              sync()
            end
            $ 440 "MoveJ"
            $ 441 "Zona_izq1" "breakAfter"
            movej(get_inverse_kin(Zona_izq1_p, qnear=Zona_izq1_q), a=1.3962634015954636, v=1.0471975511965976)
            $ 442 "Posicion_Cero" "breakAfter"
            movej(get_inverse_kin(Posicion_Cero_p, qnear=Posicion_Cero_q), a=1.3962634015954636, v=1.0471975511965976)
            $ 443 "Call Quitar_Broca_Chida"
            Quitar_Broca_Chida()
            $ 444 "Set carrusel_home=Encender"
            modbus_set_output_signal("carrusel_home", True)
            $ 445 "Wait: 1.0"
            sleep(1.0)
            $ 446 "Set carrusel_home=Apagar"
            modbus_set_output_signal("carrusel_home", False)
            $ 447 "Set mensaje_mw10=70"
            modbus_set_output_register("mensaje_mw10", 70)
            $ 448 "Wait Continuar_M30=HI"
            while (modbus_get_signal_status("Continuar_M30") == False):
              sync()
            end
            $ 449 "Wait: 1.0"
            sleep(1.0)
            $ 450 "Set mensaje_mw10=120"
            modbus_set_output_register("mensaje_mw10", 120)
            $ 451 "Wait Continuar_M30=HI"
            while (modbus_get_signal_status("Continuar_M30") == False):
              sync()
            end
            $ 452 "Wait: 1.0"
            sleep(1.0)
            $ 453 "Set carrusel_home=Encender"
            modbus_set_output_signal("carrusel_home", True)
            $ 454 "Wait: 1.0"
            sleep(1.0)
            $ 455 "Set carrusel_home=Apagar"
            modbus_set_output_signal("carrusel_home", False)
            $ 456 "Set mensaje_mw10=75"
            modbus_set_output_register("mensaje_mw10", 75)
            $ 457 "Wait Continuar_M30=HI"
            while (modbus_get_signal_status("Continuar_M30") == False):
              sync()
            end
            $ 458 "Wait: 1.0"
            sleep(1.0)
            $ 459 "Call Poner_Broca"
            Poner_Broca()
            $ 460 "broca≔1935"
            global broca=1935
            $ 461 "MoveJ"
            $ 462 "Posicion_Cero" "breakAfter"
            movej(get_inverse_kin(Posicion_Cero_p, qnear=Posicion_Cero_q), a=1.3962634015954636, v=1.0471975511965976)
            $ 463 "Zona_izq1" "breakAfter"
            movej(get_inverse_kin(Zona_izq1_p, qnear=Zona_izq1_q), a=1.3962634015954636, v=1.0471975511965976)
            $ 464 "Set mensaje_mw10=80"
            modbus_set_output_register("mensaje_mw10", 80)
            $ 465 "Wait Continuar_M30=HI"
            while (modbus_get_signal_status("Continuar_M30") == False):
              sync()
            end
            $ 466 "Wait: 1.0"
            sleep(1.0)
            $ 467 "Set mensaje_mw10=150"
            modbus_set_output_register("mensaje_mw10", 150)
            $ 468 "Wait Continuar_M30=HI"
            while (modbus_get_signal_status("Continuar_M30") == False):
              sync()
            end
            $ 469 "Wait: 1.0"
            sleep(1.0)
          end
        end
        $ 470 "barrenoActual≔barrenoActual+1"
        global barrenoActual=barrenoActual+1
      end
      $ 471 "Linea 1 a 1935"
      $ 472 "broca≔1935"
      global broca=1935
      $ 473 "Buje_inicial"
      $ 474 "Buje_Inicial≔L1B2"
      global Buje_Inicial=L1B2
      $ 475 "Buje_final"
      $ 476 "Buje_Final≔L1B1"
      global Buje_Final=L1B1
      $ 477 "barrenosTotales≔27"
      global barrenosTotales=27
      $ 478 "barrenoActual≔1"
      global barrenoActual=1
      $ 479 "Loop barrenoActual≤barrenosTotales"
      while (barrenoActual <= barrenosTotales):
        $ 480 "MoveL"
        $ 481 "bajada_broca≔p[0,0,0.009,0,0,0]"
        global bajada_broca=p[0,0,0.009,0,0,0]
        $ 482 "internos≔interpolate_pose(Buje_Inicial, Buje_Final, ((barrenoActual)-1)/((barrenosTotales)-1))"
        global internos= interpolate_pose (Buje_Inicial, Buje_Final, ((barrenoActual)-1)/((barrenosTotales)-1))
        $ 483 "Alturas"
        $ 484 "If barrenoActual≟3 or barrenoActual≟5 or barrenoActual≟7 or barrenoActual≟9 or barrenoActual≟11 or barrenoActual≟13 or barrenoActual≟15 or barrenoActual≟17 or barrenoActual≟19 or barrenoActual≟21 or barrenoActual≟23 or barrenoActual≟25 or barrenoActual≟27 or barrenoActual≟1"
        if (barrenoActual == 3  or  barrenoActual == 5  or  barrenoActual == 7  or  barrenoActual == 9  or  barrenoActual == 11  or  barrenoActual == 13  or  barrenoActual == 15  or  barrenoActual == 17  or  barrenoActual == 19  or  barrenoActual == 21  or  barrenoActual == 23  or  barrenoActual == 25  or  barrenoActual == 27  or  barrenoActual == 1):
          $ 485 "Set mensaje_mw10=200"
          modbus_set_output_register("mensaje_mw10", 200)
          $ 486 "Wait Continuar_M30=HI"
          while (modbus_get_signal_status("Continuar_M30") == False):
            sync()
          end
          $ 487 "Wait: 1.0"
          sleep(1.0)
          $ 488 "Set mensaje_mw10=150"
          modbus_set_output_register("mensaje_mw10", 150)
          $ 489 "Wait: 1.0"
          sleep(1.0)
        end
        $ 490 "MoveJ"
        $ 491 "internos" "breakAfter"
        movej(internos, a=1.3962634015954636, v=1.0471975511965976)
        $ 492 "Wait: 2.0"
        sleep(2.0)
        $ 493 "If P1h[2]<P2h[2]"
        if (P1h[2]<P2h[2]):
          $ 494 "acomodin≔(altura/(barrenosTotales-1))*(barrenoActual-1)"
          global acomodin=(altura/(barrenosTotales-1))*(barrenoActual-1)
          $ 495 "tcp_chido≔get_actual_tcp_pose()"
          global tcp_chido= get_actual_tcp_pose ()
          $ 496 "offset_bajada≔p[tcp_chido[0],tcp_chido[1],((alta-0.0095)-(acomodin/1000)),tcp_chido[3],tcp_chido[4],tcp_chido[5]]"
          global offset_bajada=p[tcp_chido[0],tcp_chido[1],((alta-0.0095)-(acomodin/1000)),tcp_chido[3],tcp_chido[4],tcp_chido[5]]
          $ 497 "MoveL"
          $ 498 "offset_bajada" "breakAfter"
          movel(offset_bajada, a=0.03, v=0.015)
        else:
          $ 499 "Else" "noBreak"
          $ 500 "acomodin≔(altura/(barrenosTotales-1))*(26-(barrenoActual-1))"
          global acomodin=(altura/(barrenosTotales-1))*(26-(barrenoActual-1))
          $ 501 "tcp_chido≔get_actual_tcp_pose()"
          global tcp_chido= get_actual_tcp_pose ()
          $ 502 "offset_bajada≔p[tcp_chido[0],tcp_chido[1],((alta-0.0095)-(acomodin/1000)),tcp_chido[3],tcp_chido[4],tcp_chido[5]]"
          global offset_bajada=p[tcp_chido[0],tcp_chido[1],((alta-0.0095)-(acomodin/1000)),tcp_chido[3],tcp_chido[4],tcp_chido[5]]
          $ 503 "MoveL"
          $ 504 "offset_bajada" "breakAfter"
          movel(offset_bajada, a=0.03, v=0.015)
        end
        $ 505 "Freemove"
        $ 506 "Wait: 2.0"
        sleep(2.0)
        $ 507 "freedrive_mode()"
        freedrive_mode()
        $ 508 "Wait: 2.5"
        sleep(2.5)
        $ 509 "end_freedrive_mode()"
        end_freedrive_mode()
        $ 510 "Wait: 0.3"
        sleep(0.3)
        $ 511 "Set CO[1]=Encender"
        set_configurable_digital_out(1, True)
        $ 512 "Wait: 1.0"
        sleep(1.0)
        $ 513 "Wait: 0.3"
        sleep(0.3)
        $ 514 "Wait: 0.3"
        sleep(0.3)
        $ 515 "Wait: 0.3"
        sleep(0.3)
        $ 516 "Loop 2 times"
        Loop_15 = 0
        while (Loop_15 < 2):
          $ 517 "Poses_taladrado≔pose_sub(get_actual_tcp_pose(), bajada_broca)"
          global Poses_taladrado= pose_sub ( get_actual_tcp_pose (), bajada_broca)
          $ 518 "Poses_taladrado" "breakAfter"
          movel(Poses_taladrado, a=0.005, v=0.001)
          $ 519 "If bajada_broca≟p[0,0,0.018,0,0,0]"
          if (bajada_broca == p[0,0,0.018,0,0,0]):
            $ 520 "num_barreno≔str_cat('Barreno: ',barrenoActual)"
            global num_barreno=str_cat("Barreno: ",barrenoActual)
            $ 521 "tcp_actual≔get_actual_tcp_pose()"
            global tcp_actual= get_actual_tcp_pose ()
            $ 522 "X_actual≔str_cat('     X: ',tcp_actual[0])"
            global X_actual=str_cat("     X: ",tcp_actual[0])
            $ 523 "Y_actual≔str_cat('     Y: ',tcp_actual[1])"
            global Y_actual=str_cat("     Y: ",tcp_actual[1])
            $ 524 "pos_barreno≔str_cat(X_actual,Y_actual)"
            global pos_barreno=str_cat(X_actual,Y_actual)
            $ 525 "textmsg(num_barreno,pos_barreno)"
            textmsg(num_barreno,pos_barreno)
          end
          $ 526 "Poses_taladrado≔pose_add(get_actual_tcp_pose(), bajada_broca)"
          global Poses_taladrado= pose_add ( get_actual_tcp_pose (), bajada_broca)
          $ 527 "Poses_taladrado" "breakAfter"
          movel(Poses_taladrado, a=0.01, v=0.01)
          $ 528 "bajada_broca≔pose_add(bajada_broca, p[0,0,0.009,0,0,0])"
          global bajada_broca= pose_add (bajada_broca, p[0,0,0.009,0,0,0])
          Loop_15 = Loop_15 + 1
        end
        $ 529 "Direction: Base Z+"
        global move_thread_flag_529=0
        thread move_thread_529():
          enter_critical
          move_thread_flag_529 = 1
          local towardsPos=calculate_point_to_move_towards(p[0.0,0.0,0.0,0.0,0.0,0.0], [0.0,0.0,1.0], 0.05)
          movel(towardsPos, a=0.04, v=0.03)
          move_thread_flag_529 = 2
          exit_critical
        end
        move_thread_flag_529 = 0
        move_thread_han_529 = run move_thread_529()
        while (True):
          sleep(1.0E-10)
          if (move_thread_flag_529 > 1):
            join move_thread_han_529
            $ 530 "Until (distance)"
            break
          end
          sync()
        end
        $ 531 "MoveJ"
        $ 532 "internos" "breakAfter"
        movej(internos, a=1.3962634015954636, v=1.0471975511965976)
        $ 533 "Wait: 0.3"
        sleep(0.3)
        $ 534 "Set CO[1]=Apagar"
        set_configurable_digital_out(1, False)
        $ 535 "Wait: 0.3"
        sleep(0.3)
        $ 536 "If barrenoActual≟13 or barrenoActual≟27"
        if (barrenoActual == 13  or  barrenoActual == 27):
          $ 537 "Direction: Base Z+"
          global move_thread_flag_537=0
          thread move_thread_537():
            enter_critical
            move_thread_flag_537 = 1
            local towardsPos=calculate_point_to_move_towards(p[0.0,0.0,0.0,0.0,0.0,0.0], [0.0,0.0,1.0], 0.03)
            movel(towardsPos, a=1.2, v=0.25)
            move_thread_flag_537 = 2
            exit_critical
          end
          move_thread_flag_537 = 0
          move_thread_han_537 = run move_thread_537()
          while (True):
            sleep(1.0E-10)
            if (move_thread_flag_537 > 1):
              join move_thread_han_537
              $ 538 "Until (distance)"
              break
            end
            sync()
          end
          $ 539 "MoveJ"
          $ 540 "Zona_izq1" "breakAfter"
          movej(get_inverse_kin(Zona_izq1_p, qnear=Zona_izq1_q), a=1.3962634015954636, v=1.0471975511965976)
          $ 541 "Posicion_Cero" "breakAfter"
          movej(get_inverse_kin(Posicion_Cero_p, qnear=Posicion_Cero_q), a=1.3962634015954636, v=1.0471975511965976)
          $ 542 "Call Quitar_Broca_Chida"
          Quitar_Broca_Chida()
          $ 543 "Call Poner_Broca"
          Poner_Broca()
          $ 544 "MoveJ"
          $ 545 "Posicion_Cero" "breakAfter"
          movej(get_inverse_kin(Posicion_Cero_p, qnear=Posicion_Cero_q), a=1.3962634015954636, v=1.0471975511965976)
          $ 546 "Zona_izq1" "breakAfter"
          movej(get_inverse_kin(Zona_izq1_p, qnear=Zona_izq1_q), a=1.3962634015954636, v=1.0471975511965976)
        end
        $ 547 "barrenoActual≔barrenoActual+1"
        global barrenoActual=barrenoActual+1
      end
      $ 548 "Linea 2 a 1935"
      $ 549 "broca≔1935"
      global broca=1935
      $ 550 "Buje_inicial"
      $ 551 "Buje_Inicial≔L2B2"
      global Buje_Inicial=L2B2
      $ 552 "Buje_final"
      $ 553 "Buje_Final≔L2B1"
      global Buje_Final=L2B1
      $ 554 "barrenosTotales≔27"
      global barrenosTotales=27
      $ 555 "barrenoActual≔1"
      global barrenoActual=1
      $ 556 "Loop barrenoActual≤barrenosTotales"
      while (barrenoActual <= barrenosTotales):
        $ 557 "MoveL"
        $ 558 "bajada_broca≔p[0,0,0.009,0,0,0]"
        global bajada_broca=p[0,0,0.009,0,0,0]
        $ 559 "internos≔interpolate_pose(Buje_Inicial, Buje_Final, ((barrenoActual)-1)/((barrenosTotales)-1))"
        global internos= interpolate_pose (Buje_Inicial, Buje_Final, ((barrenoActual)-1)/((barrenosTotales)-1))
        $ 560 "Alturas"
        $ 561 "If barrenoActual≟3 or barrenoActual≟5 or barrenoActual≟7 or barrenoActual≟9 or barrenoActual≟11 or barrenoActual≟13 or barrenoActual≟15 or barrenoActual≟17 or barrenoActual≟19 or barrenoActual≟21 or barrenoActual≟23 or barrenoActual≟25 or barrenoActual≟27 or barrenoActual≟1"
        if (barrenoActual == 3  or  barrenoActual == 5  or  barrenoActual == 7  or  barrenoActual == 9  or  barrenoActual == 11  or  barrenoActual == 13  or  barrenoActual == 15  or  barrenoActual == 17  or  barrenoActual == 19  or  barrenoActual == 21  or  barrenoActual == 23  or  barrenoActual == 25  or  barrenoActual == 27  or  barrenoActual == 1):
          $ 562 "Set mensaje_mw10=200"
          modbus_set_output_register("mensaje_mw10", 200)
          $ 563 "Wait Continuar_M30=HI"
          while (modbus_get_signal_status("Continuar_M30") == False):
            sync()
          end
          $ 564 "Wait: 1.0"
          sleep(1.0)
          $ 565 "Set mensaje_mw10=150"
          modbus_set_output_register("mensaje_mw10", 150)
          $ 566 "Wait: 1.0"
          sleep(1.0)
        end
        $ 567 "MoveJ"
        $ 568 "internos" "breakAfter"
        movej(internos, a=1.3962634015954636, v=1.0471975511965976)
        $ 569 "Wait: 2.0"
        sleep(2.0)
        $ 570 "If P1h[2]<P2h[2]"
        if (P1h[2]<P2h[2]):
          $ 571 "acomodin≔(altura/(barrenosTotales-1))*(barrenoActual-1)"
          global acomodin=(altura/(barrenosTotales-1))*(barrenoActual-1)
          $ 572 "tcp_chido≔get_actual_tcp_pose()"
          global tcp_chido= get_actual_tcp_pose ()
          $ 573 "offset_bajada≔p[tcp_chido[0],tcp_chido[1],((alta-0.0095)-(acomodin/1000)),tcp_chido[3],tcp_chido[4],tcp_chido[5]]"
          global offset_bajada=p[tcp_chido[0],tcp_chido[1],((alta-0.0095)-(acomodin/1000)),tcp_chido[3],tcp_chido[4],tcp_chido[5]]
          $ 574 "MoveL"
          $ 575 "offset_bajada" "breakAfter"
          movel(offset_bajada, a=0.03, v=0.015)
        else:
          $ 576 "Else" "noBreak"
          $ 577 "acomodin≔(altura/(barrenosTotales-1))*(26-(barrenoActual-1))"
          global acomodin=(altura/(barrenosTotales-1))*(26-(barrenoActual-1))
          $ 578 "tcp_chido≔get_actual_tcp_pose()"
          global tcp_chido= get_actual_tcp_pose ()
          $ 579 "offset_bajada≔p[tcp_chido[0],tcp_chido[1],((alta-0.0095)-(acomodin/1000)),tcp_chido[3],tcp_chido[4],tcp_chido[5]]"
          global offset_bajada=p[tcp_chido[0],tcp_chido[1],((alta-0.0095)-(acomodin/1000)),tcp_chido[3],tcp_chido[4],tcp_chido[5]]
          $ 580 "MoveL"
          $ 581 "offset_bajada" "breakAfter"
          movel(offset_bajada, a=0.03, v=0.015)
        end
        $ 582 "Freemove"
        $ 583 "Wait: 2.0"
        sleep(2.0)
        $ 584 "freedrive_mode()"
        freedrive_mode()
        $ 585 "Wait: 2.5"
        sleep(2.5)
        $ 586 "end_freedrive_mode()"
        end_freedrive_mode()
        $ 587 "Wait: 0.3"
        sleep(0.3)
        $ 588 "Set CO[1]=Encender"
        set_configurable_digital_out(1, True)
        $ 589 "Wait: 1.0"
        sleep(1.0)
        $ 590 "Wait: 0.3"
        sleep(0.3)
        $ 591 "Wait: 0.3"
        sleep(0.3)
        $ 592 "Wait: 0.3"
        sleep(0.3)
        $ 593 "Loop 2 times"
        Loop_17 = 0
        while (Loop_17 < 2):
          $ 594 "Poses_taladrado≔pose_sub(get_actual_tcp_pose(), bajada_broca)"
          global Poses_taladrado= pose_sub ( get_actual_tcp_pose (), bajada_broca)
          $ 595 "Poses_taladrado" "breakAfter"
          movel(Poses_taladrado, a=0.005, v=0.001)
          $ 596 "If bajada_broca≟p[0,0,0.018,0,0,0]"
          if (bajada_broca == p[0,0,0.018,0,0,0]):
            $ 597 "num_barreno≔str_cat('Barreno: ',barrenoActual)"
            global num_barreno=str_cat("Barreno: ",barrenoActual)
            $ 598 "tcp_actual≔get_actual_tcp_pose()"
            global tcp_actual= get_actual_tcp_pose ()
            $ 599 "X_actual≔str_cat('     X: ',tcp_actual[0])"
            global X_actual=str_cat("     X: ",tcp_actual[0])
            $ 600 "Y_actual≔str_cat('     Y: ',tcp_actual[1])"
            global Y_actual=str_cat("     Y: ",tcp_actual[1])
            $ 601 "pos_barreno≔str_cat(X_actual,Y_actual)"
            global pos_barreno=str_cat(X_actual,Y_actual)
            $ 602 "textmsg(num_barreno,pos_barreno)"
            textmsg(num_barreno,pos_barreno)
          end
          $ 603 "Poses_taladrado≔pose_add(get_actual_tcp_pose(), bajada_broca)"
          global Poses_taladrado= pose_add ( get_actual_tcp_pose (), bajada_broca)
          $ 604 "Poses_taladrado" "breakAfter"
          movel(Poses_taladrado, a=0.01, v=0.01)
          $ 605 "bajada_broca≔pose_add(bajada_broca, p[0,0,0.009,0,0,0])"
          global bajada_broca= pose_add (bajada_broca, p[0,0,0.009,0,0,0])
          Loop_17 = Loop_17 + 1
        end
        $ 606 "Direction: Base Z+"
        global move_thread_flag_606=0
        thread move_thread_606():
          enter_critical
          move_thread_flag_606 = 1
          local towardsPos=calculate_point_to_move_towards(p[0.0,0.0,0.0,0.0,0.0,0.0], [0.0,0.0,1.0], 0.05)
          movel(towardsPos, a=0.04, v=0.03)
          move_thread_flag_606 = 2
          exit_critical
        end
        move_thread_flag_606 = 0
        move_thread_han_606 = run move_thread_606()
        while (True):
          sleep(1.0E-10)
          if (move_thread_flag_606 > 1):
            join move_thread_han_606
            $ 607 "Until (distance)"
            break
          end
          sync()
        end
        $ 608 "MoveJ"
        $ 609 "internos" "breakAfter"
        movej(internos, a=1.3962634015954636, v=1.0471975511965976)
        $ 610 "Wait: 0.3"
        sleep(0.3)
        $ 611 "Set CO[1]=Apagar"
        set_configurable_digital_out(1, False)
        $ 612 "Wait: 0.3"
        sleep(0.3)
        $ 613 "If barrenoActual≟13"
        if (barrenoActual == 13):
          $ 614 "Direction: Base Z+"
          global move_thread_flag_614=0
          thread move_thread_614():
            enter_critical
            move_thread_flag_614 = 1
            local towardsPos=calculate_point_to_move_towards(p[0.0,0.0,0.0,0.0,0.0,0.0], [0.0,0.0,1.0], 0.03)
            movel(towardsPos, a=1.2, v=0.25)
            move_thread_flag_614 = 2
            exit_critical
          end
          move_thread_flag_614 = 0
          move_thread_han_614 = run move_thread_614()
          while (True):
            sleep(1.0E-10)
            if (move_thread_flag_614 > 1):
              join move_thread_han_614
              $ 615 "Until (distance)"
              break
            end
            sync()
          end
          $ 616 "MoveJ"
          $ 617 "Zona_izq1" "breakAfter"
          movej(get_inverse_kin(Zona_izq1_p, qnear=Zona_izq1_q), a=1.3962634015954636, v=1.0471975511965976)
          $ 618 "Posicion_Cero" "breakAfter"
          movej(get_inverse_kin(Posicion_Cero_p, qnear=Posicion_Cero_q), a=1.3962634015954636, v=1.0471975511965976)
          $ 619 "Call Quitar_Broca_Chida"
          Quitar_Broca_Chida()
          $ 620 "Call Poner_Broca"
          Poner_Broca()
          $ 621 "MoveJ"
          $ 622 "Posicion_Cero" "breakAfter"
          movej(get_inverse_kin(Posicion_Cero_p, qnear=Posicion_Cero_q), a=1.3962634015954636, v=1.0471975511965976)
          $ 623 "Zona_izq1" "breakAfter"
          movej(get_inverse_kin(Zona_izq1_p, qnear=Zona_izq1_q), a=1.3962634015954636, v=1.0471975511965976)
        else:
          $ 624 "ElseIf barrenoActual≟27"
          if (barrenoActual == 27):
            $ 625 "Direction: Base Z+"
            global move_thread_flag_625=0
            thread move_thread_625():
              enter_critical
              move_thread_flag_625 = 1
              local towardsPos=calculate_point_to_move_towards(p[0.0,0.0,0.0,0.0,0.0,0.0], [0.0,0.0,1.0], 0.03)
              movel(towardsPos, a=1.2, v=0.25)
              move_thread_flag_625 = 2
              exit_critical
            end
            move_thread_flag_625 = 0
            move_thread_han_625 = run move_thread_625()
            while (True):
              sleep(1.0E-10)
              if (move_thread_flag_625 > 1):
                join move_thread_han_625
                $ 626 "Until (distance)"
                break
              end
              sync()
            end
            $ 627 "MoveJ"
            $ 628 "Zona_izq1" "breakAfter"
            movej(get_inverse_kin(Zona_izq1_p, qnear=Zona_izq1_q), a=1.3962634015954636, v=1.0471975511965976)
            $ 629 "Posicion_Cero" "breakAfter"
            movej(get_inverse_kin(Posicion_Cero_p, qnear=Posicion_Cero_q), a=1.3962634015954636, v=1.0471975511965976)
            $ 630 "Call Quitar_Broca_Chida"
            Quitar_Broca_Chida()
            $ 631 "Set carrusel_home=Encender"
            modbus_set_output_signal("carrusel_home", True)
            $ 632 "Wait: 1.0"
            sleep(1.0)
            $ 633 "Set carrusel_home=Apagar"
            modbus_set_output_signal("carrusel_home", False)
            $ 634 "Set mensaje_mw10=85"
            modbus_set_output_register("mensaje_mw10", 85)
            $ 635 "Wait Continuar_M30=HI"
            while (modbus_get_signal_status("Continuar_M30") == False):
              sync()
            end
            $ 636 "Wait: 1.0"
            sleep(1.0)
            $ 637 "Set mensaje_mw10=120"
            modbus_set_output_register("mensaje_mw10", 120)
            $ 638 "Wait Continuar_M30=HI"
            while (modbus_get_signal_status("Continuar_M30") == False):
              sync()
            end
            $ 639 "Wait: 1.0"
            sleep(1.0)
            $ 640 "Set carrusel_home=Encender"
            modbus_set_output_signal("carrusel_home", True)
            $ 641 "Wait: 1.0"
            sleep(1.0)
            $ 642 "Set carrusel_home=Apagar"
            modbus_set_output_signal("carrusel_home", False)
            $ 643 "Set mensaje_mw10=90"
            modbus_set_output_register("mensaje_mw10", 90)
            $ 644 "Wait Continuar_M30=HI"
            while (modbus_get_signal_status("Continuar_M30") == False):
              sync()
            end
            $ 645 "Wait: 1.0"
            sleep(1.0)
            $ 646 "Call Poner_Broca"
            Poner_Broca()
            $ 647 "broca≔217"
            global broca=217
            $ 648 "MoveJ"
            $ 649 "Posicion_Cero" "breakAfter"
            movej(get_inverse_kin(Posicion_Cero_p, qnear=Posicion_Cero_q), a=1.3962634015954636, v=1.0471975511965976)
            $ 650 "Zona_izq1" "breakAfter"
            movej(get_inverse_kin(Zona_izq1_p, qnear=Zona_izq1_q), a=1.3962634015954636, v=1.0471975511965976)
            $ 651 "Set mensaje_mw10=95"
            modbus_set_output_register("mensaje_mw10", 95)
            $ 652 "Wait Continuar_M30=HI"
            while (modbus_get_signal_status("Continuar_M30") == False):
              sync()
            end
            $ 653 "Wait: 1.0"
            sleep(1.0)
            $ 654 "Set mensaje_mw10=150"
            modbus_set_output_register("mensaje_mw10", 150)
            $ 655 "Wait Continuar_M30=HI"
            while (modbus_get_signal_status("Continuar_M30") == False):
              sync()
            end
            $ 656 "Wait: 1.0"
            sleep(1.0)
          end
        end
        $ 657 "barrenoActual≔barrenoActual+1"
        global barrenoActual=barrenoActual+1
      end
      $ 658 "Linea 1 a 217"
      $ 659 "broca≔217"
      global broca=217
      $ 660 "Buje_inicial"
      $ 661 "Buje_Inicial≔L1B2"
      global Buje_Inicial=L1B2
      $ 662 "Buje_final"
      $ 663 "Buje_Final≔L1B1"
      global Buje_Final=L1B1
      $ 664 "barrenosTotales≔27"
      global barrenosTotales=27
      $ 665 "barrenoActual≔1"
      global barrenoActual=1
      $ 666 "Loop barrenoActual≤barrenosTotales"
      while (barrenoActual <= barrenosTotales):
        $ 667 "MoveL"
        $ 668 "bajada_broca≔p[0,0,0.018,0,0,0]"
        global bajada_broca=p[0,0,0.018,0,0,0]
        $ 669 "internos≔interpolate_pose(Buje_Inicial, Buje_Final, ((barrenoActual)-1)/((barrenosTotales)-1))"
        global internos= interpolate_pose (Buje_Inicial, Buje_Final, ((barrenoActual)-1)/((barrenosTotales)-1))
        $ 670 "Alturas"
        $ 671 "If barrenoActual≟3 or barrenoActual≟5 or barrenoActual≟7 or barrenoActual≟9 or barrenoActual≟11 or barrenoActual≟13 or barrenoActual≟15 or barrenoActual≟17 or barrenoActual≟19 or barrenoActual≟21 or barrenoActual≟23 or barrenoActual≟25 or barrenoActual≟27 or barrenoActual≟1"
        if (barrenoActual == 3  or  barrenoActual == 5  or  barrenoActual == 7  or  barrenoActual == 9  or  barrenoActual == 11  or  barrenoActual == 13  or  barrenoActual == 15  or  barrenoActual == 17  or  barrenoActual == 19  or  barrenoActual == 21  or  barrenoActual == 23  or  barrenoActual == 25  or  barrenoActual == 27  or  barrenoActual == 1):
          $ 672 "Set mensaje_mw10=200"
          modbus_set_output_register("mensaje_mw10", 200)
          $ 673 "Wait Continuar_M30=HI"
          while (modbus_get_signal_status("Continuar_M30") == False):
            sync()
          end
          $ 674 "Wait: 1.0"
          sleep(1.0)
          $ 675 "Set mensaje_mw10=150"
          modbus_set_output_register("mensaje_mw10", 150)
          $ 676 "Wait: 1.0"
          sleep(1.0)
        end
        $ 677 "MoveJ"
        $ 678 "internos" "breakAfter"
        movej(internos, a=1.3962634015954636, v=1.0471975511965976)
        $ 679 "Wait: 2.0"
        sleep(2.0)
        $ 680 "If P1h[2]<P2h[2]"
        if (P1h[2]<P2h[2]):
          $ 681 "acomodin≔(altura/(barrenosTotales-1))*(barrenoActual-1)"
          global acomodin=(altura/(barrenosTotales-1))*(barrenoActual-1)
          $ 682 "tcp_chido≔get_actual_tcp_pose()"
          global tcp_chido= get_actual_tcp_pose ()
          $ 683 "offset_bajada≔p[tcp_chido[0],tcp_chido[1],((alta-0.0095)-(acomodin/1000)),tcp_chido[3],tcp_chido[4],tcp_chido[5]]"
          global offset_bajada=p[tcp_chido[0],tcp_chido[1],((alta-0.0095)-(acomodin/1000)),tcp_chido[3],tcp_chido[4],tcp_chido[5]]
          $ 684 "MoveL"
          $ 685 "offset_bajada" "breakAfter"
          movel(offset_bajada, a=0.03, v=0.015)
        else:
          $ 686 "Else" "noBreak"
          $ 687 "acomodin≔(altura/(barrenosTotales-1))*(26-(barrenoActual-1))"
          global acomodin=(altura/(barrenosTotales-1))*(26-(barrenoActual-1))
          $ 688 "tcp_chido≔get_actual_tcp_pose()"
          global tcp_chido= get_actual_tcp_pose ()
          $ 689 "offset_bajada≔p[tcp_chido[0],tcp_chido[1],((alta-0.0095)-(acomodin/1000)),tcp_chido[3],tcp_chido[4],tcp_chido[5]]"
          global offset_bajada=p[tcp_chido[0],tcp_chido[1],((alta-0.0095)-(acomodin/1000)),tcp_chido[3],tcp_chido[4],tcp_chido[5]]
          $ 690 "MoveL"
          $ 691 "offset_bajada" "breakAfter"
          movel(offset_bajada, a=0.03, v=0.015)
        end
        $ 692 "Freemove"
        $ 693 "Wait: 2.0"
        sleep(2.0)
        $ 694 "freedrive_mode()"
        freedrive_mode()
        $ 695 "Wait: 2.5"
        sleep(2.5)
        $ 696 "end_freedrive_mode()"
        end_freedrive_mode()
        $ 697 "Wait: 0.3"
        sleep(0.3)
        $ 698 "Set CO[1]=Encender"
        set_configurable_digital_out(1, True)
        $ 699 "Wait: 1.0"
        sleep(1.0)
        $ 700 "Wait: 0.3"
        sleep(0.3)
        $ 701 "Wait: 0.3"
        sleep(0.3)
        $ 702 "Wait: 0.3"
        sleep(0.3)
        $ 703 "Loop 1 times"
        Loop_19 = 0
        while (Loop_19 < 1):
          $ 704 "Poses_taladrado≔pose_sub(get_actual_tcp_pose(), bajada_broca)"
          global Poses_taladrado= pose_sub ( get_actual_tcp_pose (), bajada_broca)
          $ 705 "Poses_taladrado" "breakAfter"
          movel(Poses_taladrado, a=0.005, v=0.001)
          $ 706 "If bajada_broca≟p[0,0,0.018,0,0,0]"
          if (bajada_broca == p[0,0,0.018,0,0,0]):
            $ 707 "num_barreno≔str_cat('Barreno: ',barrenoActual)"
            global num_barreno=str_cat("Barreno: ",barrenoActual)
            $ 708 "tcp_actual≔get_actual_tcp_pose()"
            global tcp_actual= get_actual_tcp_pose ()
            $ 709 "X_actual≔str_cat('     X: ',tcp_actual[0])"
            global X_actual=str_cat("     X: ",tcp_actual[0])
            $ 710 "Y_actual≔str_cat('     Y: ',tcp_actual[1])"
            global Y_actual=str_cat("     Y: ",tcp_actual[1])
            $ 711 "pos_barreno≔str_cat(X_actual,Y_actual)"
            global pos_barreno=str_cat(X_actual,Y_actual)
            $ 712 "textmsg(num_barreno,pos_barreno)"
            textmsg(num_barreno,pos_barreno)
          end
          $ 713 "Poses_taladrado≔pose_add(get_actual_tcp_pose(), bajada_broca)"
          global Poses_taladrado= pose_add ( get_actual_tcp_pose (), bajada_broca)
          $ 714 "Poses_taladrado" "breakAfter"
          movel(Poses_taladrado, a=0.01, v=0.01)
          $ 715 "bajada_broca≔pose_add(bajada_broca, p[0,0,0.018,0,0,0])"
          global bajada_broca= pose_add (bajada_broca, p[0,0,0.018,0,0,0])
          Loop_19 = Loop_19 + 1
        end
        $ 716 "Direction: Base Z+"
        global move_thread_flag_716=0
        thread move_thread_716():
          enter_critical
          move_thread_flag_716 = 1
          local towardsPos=calculate_point_to_move_towards(p[0.0,0.0,0.0,0.0,0.0,0.0], [0.0,0.0,1.0], 0.05)
          movel(towardsPos, a=0.04, v=0.03)
          move_thread_flag_716 = 2
          exit_critical
        end
        move_thread_flag_716 = 0
        move_thread_han_716 = run move_thread_716()
        while (True):
          sleep(1.0E-10)
          if (move_thread_flag_716 > 1):
            join move_thread_han_716
            $ 717 "Until (distance)"
            break
          end
          sync()
        end
        $ 718 "MoveJ"
        $ 719 "internos" "breakAfter"
        movej(internos, a=1.3962634015954636, v=1.0471975511965976)
        $ 720 "Wait: 0.3"
        sleep(0.3)
        $ 721 "Set CO[1]=Apagar"
        set_configurable_digital_out(1, False)
        $ 722 "Wait: 0.3"
        sleep(0.3)
        $ 723 "If barrenoActual≟13 or barrenoActual≟27"
        if (barrenoActual == 13  or  barrenoActual == 27):
          $ 724 "Direction: Base Z+"
          global move_thread_flag_724=0
          thread move_thread_724():
            enter_critical
            move_thread_flag_724 = 1
            local towardsPos=calculate_point_to_move_towards(p[0.0,0.0,0.0,0.0,0.0,0.0], [0.0,0.0,1.0], 0.03)
            movel(towardsPos, a=1.2, v=0.25)
            move_thread_flag_724 = 2
            exit_critical
          end
          move_thread_flag_724 = 0
          move_thread_han_724 = run move_thread_724()
          while (True):
            sleep(1.0E-10)
            if (move_thread_flag_724 > 1):
              join move_thread_han_724
              $ 725 "Until (distance)"
              break
            end
            sync()
          end
          $ 726 "MoveJ"
          $ 727 "Zona_izq1" "breakAfter"
          movej(get_inverse_kin(Zona_izq1_p, qnear=Zona_izq1_q), a=1.3962634015954636, v=1.0471975511965976)
          $ 728 "Posicion_Cero" "breakAfter"
          movej(get_inverse_kin(Posicion_Cero_p, qnear=Posicion_Cero_q), a=1.3962634015954636, v=1.0471975511965976)
          $ 729 "Call Quitar_Broca_Chida"
          Quitar_Broca_Chida()
          $ 730 "Call Poner_Broca"
          Poner_Broca()
          $ 731 "MoveJ"
          $ 732 "Posicion_Cero" "breakAfter"
          movej(get_inverse_kin(Posicion_Cero_p, qnear=Posicion_Cero_q), a=1.3962634015954636, v=1.0471975511965976)
          $ 733 "Zona_izq1" "breakAfter"
          movej(get_inverse_kin(Zona_izq1_p, qnear=Zona_izq1_q), a=1.3962634015954636, v=1.0471975511965976)
        end
        $ 734 "barrenoActual≔barrenoActual+1"
        global barrenoActual=barrenoActual+1
      end
      $ 735 "Linea 2 a 217"
      $ 736 "broca≔217"
      global broca=217
      $ 737 "Buje_inicial"
      $ 738 "Buje_Inicial≔L2B2"
      global Buje_Inicial=L2B2
      $ 739 "Buje_final"
      $ 740 "Buje_Final≔L2B1"
      global Buje_Final=L2B1
      $ 741 "barrenosTotales≔27"
      global barrenosTotales=27
      $ 742 "barrenoActual≔1"
      global barrenoActual=1
      $ 743 "Loop barrenoActual≤barrenosTotales"
      while (barrenoActual <= barrenosTotales):
        $ 744 "MoveL"
        $ 745 "bajada_broca≔p[0,0,0.018,0,0,0]"
        global bajada_broca=p[0,0,0.018,0,0,0]
        $ 746 "internos≔interpolate_pose(Buje_Inicial, Buje_Final, ((barrenoActual)-1)/((barrenosTotales)-1))"
        global internos= interpolate_pose (Buje_Inicial, Buje_Final, ((barrenoActual)-1)/((barrenosTotales)-1))
        $ 747 "Alturas"
        $ 748 "If barrenoActual≟3 or barrenoActual≟5 or barrenoActual≟7 or barrenoActual≟9 or barrenoActual≟11 or barrenoActual≟13 or barrenoActual≟15 or barrenoActual≟17 or barrenoActual≟19 or barrenoActual≟21 or barrenoActual≟23 or barrenoActual≟25 or barrenoActual≟27 or barrenoActual≟1"
        if (barrenoActual == 3  or  barrenoActual == 5  or  barrenoActual == 7  or  barrenoActual == 9  or  barrenoActual == 11  or  barrenoActual == 13  or  barrenoActual == 15  or  barrenoActual == 17  or  barrenoActual == 19  or  barrenoActual == 21  or  barrenoActual == 23  or  barrenoActual == 25  or  barrenoActual == 27  or  barrenoActual == 1):
          $ 749 "Set mensaje_mw10=200"
          modbus_set_output_register("mensaje_mw10", 200)
          $ 750 "Wait Continuar_M30=HI"
          while (modbus_get_signal_status("Continuar_M30") == False):
            sync()
          end
          $ 751 "Wait: 1.0"
          sleep(1.0)
          $ 752 "Set mensaje_mw10=150"
          modbus_set_output_register("mensaje_mw10", 150)
          $ 753 "Wait: 1.0"
          sleep(1.0)
        end
        $ 754 "MoveJ"
        $ 755 "internos" "breakAfter"
        movej(internos, a=1.3962634015954636, v=1.0471975511965976)
        $ 756 "Wait: 2.0"
        sleep(2.0)
        $ 757 "If P1h[2]<P2h[2]"
        if (P1h[2]<P2h[2]):
          $ 758 "acomodin≔(altura/(barrenosTotales-1))*(barrenoActual-1)"
          global acomodin=(altura/(barrenosTotales-1))*(barrenoActual-1)
          $ 759 "tcp_chido≔get_actual_tcp_pose()"
          global tcp_chido= get_actual_tcp_pose ()
          $ 760 "offset_bajada≔p[tcp_chido[0],tcp_chido[1],((alta-0.0095)-(acomodin/1000)),tcp_chido[3],tcp_chido[4],tcp_chido[5]]"
          global offset_bajada=p[tcp_chido[0],tcp_chido[1],((alta-0.0095)-(acomodin/1000)),tcp_chido[3],tcp_chido[4],tcp_chido[5]]
          $ 761 "MoveL"
          $ 762 "offset_bajada" "breakAfter"
          movel(offset_bajada, a=0.03, v=0.015)
        else:
          $ 763 "Else" "noBreak"
          $ 764 "acomodin≔(altura/(barrenosTotales-1))*(26-(barrenoActual-1))"
          global acomodin=(altura/(barrenosTotales-1))*(26-(barrenoActual-1))
          $ 765 "tcp_chido≔get_actual_tcp_pose()"
          global tcp_chido= get_actual_tcp_pose ()
          $ 766 "offset_bajada≔p[tcp_chido[0],tcp_chido[1],((alta-0.0095)-(acomodin/1000)),tcp_chido[3],tcp_chido[4],tcp_chido[5]]"
          global offset_bajada=p[tcp_chido[0],tcp_chido[1],((alta-0.0095)-(acomodin/1000)),tcp_chido[3],tcp_chido[4],tcp_chido[5]]
          $ 767 "MoveL"
          $ 768 "offset_bajada" "breakAfter"
          movel(offset_bajada, a=0.03, v=0.015)
        end
        $ 769 "Freemove"
        $ 770 "Wait: 2.0"
        sleep(2.0)
        $ 771 "freedrive_mode()"
        freedrive_mode()
        $ 772 "Wait: 2.5"
        sleep(2.5)
        $ 773 "end_freedrive_mode()"
        end_freedrive_mode()
        $ 774 "Wait: 0.3"
        sleep(0.3)
        $ 775 "Set CO[1]=Encender"
        set_configurable_digital_out(1, True)
        $ 776 "Wait: 1.0"
        sleep(1.0)
        $ 777 "Wait: 0.3"
        sleep(0.3)
        $ 778 "Wait: 0.3"
        sleep(0.3)
        $ 779 "Wait: 0.3"
        sleep(0.3)
        $ 780 "Loop 1 times"
        Loop_21 = 0
        while (Loop_21 < 1):
          $ 781 "Poses_taladrado≔pose_sub(get_actual_tcp_pose(), bajada_broca)"
          global Poses_taladrado= pose_sub ( get_actual_tcp_pose (), bajada_broca)
          $ 782 "Poses_taladrado" "breakAfter"
          movel(Poses_taladrado, a=0.005, v=0.001)
          $ 783 "If bajada_broca≟p[0,0,0.018,0,0,0]"
          if (bajada_broca == p[0,0,0.018,0,0,0]):
            $ 784 "num_barreno≔str_cat('Barreno: ',barrenoActual)"
            global num_barreno=str_cat("Barreno: ",barrenoActual)
            $ 785 "tcp_actual≔get_actual_tcp_pose()"
            global tcp_actual= get_actual_tcp_pose ()
            $ 786 "X_actual≔str_cat('     X: ',tcp_actual[0])"
            global X_actual=str_cat("     X: ",tcp_actual[0])
            $ 787 "Y_actual≔str_cat('     Y: ',tcp_actual[1])"
            global Y_actual=str_cat("     Y: ",tcp_actual[1])
            $ 788 "pos_barreno≔str_cat(X_actual,Y_actual)"
            global pos_barreno=str_cat(X_actual,Y_actual)
            $ 789 "textmsg(num_barreno,pos_barreno)"
            textmsg(num_barreno,pos_barreno)
          end
          $ 790 "Poses_taladrado≔pose_add(get_actual_tcp_pose(), bajada_broca)"
          global Poses_taladrado= pose_add ( get_actual_tcp_pose (), bajada_broca)
          $ 791 "Poses_taladrado" "breakAfter"
          movel(Poses_taladrado, a=0.01, v=0.01)
          $ 792 "bajada_broca≔pose_add(bajada_broca, p[0,0,0.018,0,0,0])"
          global bajada_broca= pose_add (bajada_broca, p[0,0,0.018,0,0,0])
          Loop_21 = Loop_21 + 1
        end
        $ 793 "Direction: Base Z+"
        global move_thread_flag_793=0
        thread move_thread_793():
          enter_critical
          move_thread_flag_793 = 1
          local towardsPos=calculate_point_to_move_towards(p[0.0,0.0,0.0,0.0,0.0,0.0], [0.0,0.0,1.0], 0.05)
          movel(towardsPos, a=0.04, v=0.03)
          move_thread_flag_793 = 2
          exit_critical
        end
        move_thread_flag_793 = 0
        move_thread_han_793 = run move_thread_793()
        while (True):
          sleep(1.0E-10)
          if (move_thread_flag_793 > 1):
            join move_thread_han_793
            $ 794 "Until (distance)"
            break
          end
          sync()
        end
        $ 795 "MoveJ"
        $ 796 "internos" "breakAfter"
        movej(internos, a=1.3962634015954636, v=1.0471975511965976)
        $ 797 "Wait: 0.3"
        sleep(0.3)
        $ 798 "Set CO[1]=Apagar"
        set_configurable_digital_out(1, False)
        $ 799 "Wait: 0.3"
        sleep(0.3)
        $ 800 "If barrenoActual≟13"
        if (barrenoActual == 13):
          $ 801 "Direction: Base Z+"
          global move_thread_flag_801=0
          thread move_thread_801():
            enter_critical
            move_thread_flag_801 = 1
            local towardsPos=calculate_point_to_move_towards(p[0.0,0.0,0.0,0.0,0.0,0.0], [0.0,0.0,1.0], 0.03)
            movel(towardsPos, a=1.2, v=0.25)
            move_thread_flag_801 = 2
            exit_critical
          end
          move_thread_flag_801 = 0
          move_thread_han_801 = run move_thread_801()
          while (True):
            sleep(1.0E-10)
            if (move_thread_flag_801 > 1):
              join move_thread_han_801
              $ 802 "Until (distance)"
              break
            end
            sync()
          end
          $ 803 "MoveJ"
          $ 804 "Zona_izq1" "breakAfter"
          movej(get_inverse_kin(Zona_izq1_p, qnear=Zona_izq1_q), a=1.3962634015954636, v=1.0471975511965976)
          $ 805 "Posicion_Cero" "breakAfter"
          movej(get_inverse_kin(Posicion_Cero_p, qnear=Posicion_Cero_q), a=1.3962634015954636, v=1.0471975511965976)
          $ 806 "Call Quitar_Broca_Chida"
          Quitar_Broca_Chida()
          $ 807 "Call Poner_Broca"
          Poner_Broca()
          $ 808 "MoveJ"
          $ 809 "Posicion_Cero" "breakAfter"
          movej(get_inverse_kin(Posicion_Cero_p, qnear=Posicion_Cero_q), a=1.3962634015954636, v=1.0471975511965976)
          $ 810 "Zona_izq1" "breakAfter"
          movej(get_inverse_kin(Zona_izq1_p, qnear=Zona_izq1_q), a=1.3962634015954636, v=1.0471975511965976)
        else:
          $ 811 "ElseIf barrenoActual≟27"
          if (barrenoActual == 27):
            $ 812 "Direction: Base Z+"
            global move_thread_flag_812=0
            thread move_thread_812():
              enter_critical
              move_thread_flag_812 = 1
              local towardsPos=calculate_point_to_move_towards(p[0.0,0.0,0.0,0.0,0.0,0.0], [0.0,0.0,1.0], 0.03)
              movel(towardsPos, a=1.2, v=0.25)
              move_thread_flag_812 = 2
              exit_critical
            end
            move_thread_flag_812 = 0
            move_thread_han_812 = run move_thread_812()
            while (True):
              sleep(1.0E-10)
              if (move_thread_flag_812 > 1):
                join move_thread_han_812
                $ 813 "Until (distance)"
                break
              end
              sync()
            end
            $ 814 "MoveJ"
            $ 815 "Zona_izq1" "breakAfter"
            movej(get_inverse_kin(Zona_izq1_p, qnear=Zona_izq1_q), a=1.3962634015954636, v=1.0471975511965976)
            $ 816 "Posicion_Cero" "breakAfter"
            movej(get_inverse_kin(Posicion_Cero_p, qnear=Posicion_Cero_q), a=1.3962634015954636, v=1.0471975511965976)
            $ 817 "Call Quitar_Broca_Chida"
            Quitar_Broca_Chida()
            $ 818 "Set carrusel_home=Encender"
            modbus_set_output_signal("carrusel_home", True)
            $ 819 "Wait: 1.0"
            sleep(1.0)
            $ 820 "Set carrusel_home=Apagar"
            modbus_set_output_signal("carrusel_home", False)
            $ 821 "Set mensaje_mw10=120"
            modbus_set_output_register("mensaje_mw10", 120)
            $ 822 "Wait Continuar_M30=HI"
            while (modbus_get_signal_status("Continuar_M30") == False):
              sync()
            end
            $ 823 "Wait: 1.0"
            sleep(1.0)
            $ 824 "Set mensaje_mw10=100"
            modbus_set_output_register("mensaje_mw10", 100)
            $ 825 "Wait Continuar_M30=HI"
            while (modbus_get_signal_status("Continuar_M30") == False):
              sync()
            end
            $ 826 "Wait: 1.0"
            sleep(1.0)
            $ 827 "MoveJ"
            $ 828 "Traslacion_izq" "breakAfter"
            movej(get_inverse_kin(Traslacion_izq_p, qnear=Traslacion_izq_q), a=1.3962634015954636, v=1.0471975511965976)
          end
        end
        $ 829 "barrenoActual≔barrenoActual+1"
        global barrenoActual=barrenoActual+1
      end
      $ 831 "Traslacion"
      $ 832 "MoveJ"
      $ 833 "Traslacion_izq" "breakAfter"
      movej(get_inverse_kin(Traslacion_izq_p, qnear=Traslacion_izq_q), a=1.3962634015954636, v=1.0471975511965976)
      $ 834 "Set mensaje_mw10=105"
      modbus_set_output_register("mensaje_mw10", 105)
      $ 835 "Wait Continuar_M30=HI"
      while (modbus_get_signal_status("Continuar_M30") == False):
        sync()
      end
      $ 836 "Wait: 1.0"
      sleep(1.0)
      $ 837 "Set mensaje_mw10=145"
      modbus_set_output_register("mensaje_mw10", 145)
      $ 838 "Wait Continuar_M30=HI"
      while (modbus_get_signal_status("Continuar_M30") == False):
        sync()
      end
      $ 839 "Wait: 1.0"
      sleep(1.0)
      $ 840 "Set postrnas_m187=Encender"
      modbus_set_output_signal("postrnas_m187", True)
      $ 841 "Wait: 1.0"
      sleep(1.0)
      $ 842 "Set pos2_izq_m697=Encender"
      modbus_set_output_signal("pos2_izq_m697", True)
      $ 843 "Wait: 1.0"
      sleep(1.0)
      $ 844 "Set pos2_izq_m697=Apagar"
      modbus_set_output_signal("pos2_izq_m697", False)
      $ 845 "Set postrnas_m187=Apagar"
      modbus_set_output_signal("postrnas_m187", False)
      $ 846 "Wait: 5.0"
      sleep(5.0)
      $ 847 "Brocas"
      $ 848 "Set carrusel_home=Encender"
      modbus_set_output_signal("carrusel_home", True)
      $ 849 "Wait: 1.0"
      sleep(1.0)
      $ 850 "Set carrusel_home=Apagar"
      modbus_set_output_signal("carrusel_home", False)
      $ 851 "Set mensaje_mw10=40"
      modbus_set_output_register("mensaje_mw10", 40)
      $ 852 "Wait Continuar_M30=HI"
      while (modbus_get_signal_status("Continuar_M30") == False):
        sync()
      end
      $ 853 "Wait: 1.0"
      sleep(1.0)
      $ 854 "Set carrusel_home=Encender"
      modbus_set_output_signal("carrusel_home", True)
      $ 855 "Wait: 1.0"
      sleep(1.0)
      $ 856 "Set carrusel_home=Apagar"
      modbus_set_output_signal("carrusel_home", False)
      $ 857 "Set mensaje_mw10=45"
      modbus_set_output_register("mensaje_mw10", 45)
      $ 858 "Wait Continuar_M30=HI"
      while (modbus_get_signal_status("Continuar_M30") == False):
        sync()
      end
      $ 859 "Wait: 1.0"
      sleep(1.0)
      $ 860 "Call Poner_Broca"
      Poner_Broca()
      $ 861 "Offsets factor"
      $ 863 "L1B1x≔((0.09523476)/(0.09525))*(0.09523476)"
      global L1B1x=((0.09523476)/(0.09525))*(0.09523476)
      $ 864 "L1B1y≔((-0.01278382)/(-0.0127))*(-0.01278382)"
      global L1B1y=((-0.01278382)/(-0.0127))*(-0.01278382)
      $ 865 "L1B2x≔((0.75575414)/(0.75565))*(0.75575414)"
      global L1B2x=((0.75575414)/(0.75565))*(0.75575414)
      $ 866 "L1B2y≔((-0.01279398)/(-0.0127))*(-0.01279398)"
      global L1B2y=((-0.01279398)/(-0.0127))*(-0.01279398)
      $ 867 "L2B1x≔((0.09675299)/(0.09525))*(0.09675299)"
      global L2B1x=((0.09675299)/(0.09525))*(0.09675299)
      $ 868 "L2B1y≔((0.3937)/(0.3937))*(0.3937)"
      global L2B1y=((0.3937)/(0.3937))*(0.3937)
      $ 869 "L2B2x≔((0.757306777)/(0.75565))*(0.757306777)"
      global L2B2x=((0.757306777)/(0.75565))*(0.757306777)
      $ 870 "L2B2y≔((0.393684081)/(0.3937))*(0.393684081)"
      global L2B2y=((0.393684081)/(0.3937))*(0.393684081)
      $ 871 "Calibracion"
      $ 872 "Set mensaje_mw10=50"
      modbus_set_output_register("mensaje_mw10", 50)
      $ 873 "Wait Continuar_M30=HI"
      while (modbus_get_signal_status("Continuar_M30") == False):
        sync()
      end
      $ 874 "Wait: 1.0"
      sleep(1.0)
      $ 875 "MoveJ"
      $ 876 "Posicion_Cero" "breakAfter"
      movej(get_inverse_kin(Posicion_Cero_p, qnear=Posicion_Cero_q), a=1.3962634015954636, v=1.0471975511965976)
      $ 877 "Zona_izq1" "breakAfter"
      movej(get_inverse_kin(Zona_izq1_p, qnear=Zona_izq1_q), a=1.3962634015954636, v=1.0471975511965976)
      $ 878 "broca≔1645"
      global broca=1645
      $ 879 "Set mensaje_mw10=125"
      modbus_set_output_register("mensaje_mw10", 125)
      $ 880 "Wait Continuar_M30=HI"
      while (modbus_get_signal_status("Continuar_M30") == False):
        sync()
      end
      $ 881 "Wait: 1.0"
      sleep(1.0)
      $ 882 "Set mensaje_mw10=130"
      modbus_set_output_register("mensaje_mw10", 130)
      $ 883 "Wait Continuar_M30=HI"
      while (modbus_get_signal_status("Continuar_M30") == False):
        sync()
      end
      $ 884 "Wait: 1.0"
      sleep(1.0)
      $ 885 "Call Calibracion"
      Calibracion()
      $ 886 "GoNoGo"
      $ 887 "Set mensaje_mw10=55"
      modbus_set_output_register("mensaje_mw10", 55)
      $ 888 "Wait Continuar_M30=HI"
      while (modbus_get_signal_status("Continuar_M30") == False):
        sync()
      end
      $ 889 "Wait: 1.0"
      sleep(1.0)
      $ 890 "Set mensaje_mw10=60"
      modbus_set_output_register("mensaje_mw10", 60)
      $ 891 "Wait Continuar_M30=HI"
      while (modbus_get_signal_status("Continuar_M30") == False):
        sync()
      end
      $ 892 "Wait: 1.0"
      sleep(1.0)
      $ 893 "Linea1_Buje1"
      $ 894 "Xfin≔((((L1B1x)*(-1)*Xp)-(Xd)-((L1B1y)*(1/m2)))*(-1))*(1)"
      global Xfin=((((L1B1x)*(-1)*Xp)-(Xd)-((L1B1y)*(1/m2)))*(-1))*(1)
      $ 895 "Yfin≔((((L1B1y)*(-1)*Yp)-(Yd)+((L1B1x)*(-1)*m1))*(-1))*(1)"
      global Yfin=((((L1B1y)*(-1)*Yp)-(Yd)+((L1B1x)*(-1)*m1))*(-1))*(1)
      $ 896 "rotaciones≔get_actual_tcp_pose()"
      global rotaciones= get_actual_tcp_pose ()
      $ 897 "var_3≔rotaciones[3]"
      global var_3=rotaciones[3]
      $ 898 "var_4≔rotaciones[4]"
      global var_4=rotaciones[4]
      $ 899 "var_5≔rotaciones[5]"
      global var_5=rotaciones[5]
      $ 900 "If broca≟1645"
      if (broca == 1645):
        $ 901 "PosFinal≔p[Xfin-0.00208915,Yfin-0.00208915,0.15,var_3,var_4,var_5]"
        global PosFinal=p[Xfin-0.00208915,Yfin-0.00208915,0.15,var_3,var_4,var_5]
      else:
        $ 902 "ElseIf broca≟1935"
        if (broca == 1935):
          $ 903 "PosFinal≔p[Xfin-0.00245745,Yfin-0.00245745,0.15,var_3,var_4,var_5]"
          global PosFinal=p[Xfin-0.00245745,Yfin-0.00245745,0.15,var_3,var_4,var_5]
        else:
          $ 904 "ElseIf broca≟217"
          if (broca == 217):
            $ 905 "PosFinal≔p[Xfin-0.0027559,Yfin-0.0027559,0.15,var_3,var_4,var_5]"
            global PosFinal=p[Xfin-0.0027559,Yfin-0.0027559,0.15,var_3,var_4,var_5]
          end
        end
      end
      $ 906 "Buje_Final≔PosFinal"
      global Buje_Final=PosFinal
      $ 907 "MoveJ"
      $ 908 "Buje_Final" "breakAfter"
      movej(Buje_Final, a=1.3962634015954636, v=1.0471975511965976)
      $ 909 "Wait: 1.0"
      sleep(1.0)
      $ 910 "Alturas"
      $ 911 "If P1h[2]<P2h[2]"
      if (P1h[2]<P2h[2]):
        $ 912 "tcp_chido≔get_actual_tcp_pose()"
        global tcp_chido= get_actual_tcp_pose ()
        $ 913 "offset_bajada≔p[tcp_chido[0],tcp_chido[1],((alta-0.0095)-(altura/1000)),tcp_chido[3],tcp_chido[4],tcp_chido[5]]"
        global offset_bajada=p[tcp_chido[0],tcp_chido[1],((alta-0.0095)-(altura/1000)),tcp_chido[3],tcp_chido[4],tcp_chido[5]]
        $ 914 "MoveL"
        $ 915 "offset_bajada" "breakAfter"
        movel(offset_bajada, a=0.03, v=0.015)
      else:
        $ 916 "Else" "noBreak"
        $ 917 "tcp_chido≔get_actual_tcp_pose()"
        global tcp_chido= get_actual_tcp_pose ()
        $ 918 "offset_bajada≔p[tcp_chido[0],tcp_chido[1],((alta-0.0095)),tcp_chido[3],tcp_chido[4],tcp_chido[5]]"
        global offset_bajada=p[tcp_chido[0],tcp_chido[1],((alta-0.0095)),tcp_chido[3],tcp_chido[4],tcp_chido[5]]
        $ 919 "MoveL"
        $ 920 "offset_bajada" "breakAfter"
        movel(offset_bajada, a=0.03, v=0.015)
      end
      $ 921 "MoveL"
      $ 922 "Freemove"
      $ 923 "Wait: 2.0"
      sleep(2.0)
      $ 924 "freedrive_mode()"
      freedrive_mode()
      $ 925 "Wait: 2.5"
      sleep(2.5)
      $ 926 "end_freedrive_mode()"
      end_freedrive_mode()
      $ 927 "var_13≔get_actual_tcp_pose()"
      global var_13= get_actual_tcp_pose ()
      $ 928 "var_13≔p[var_13[0]*1000,var_13[1]*1000,420,420,420,420]"
      global var_13=p[var_13[0]*1000,var_13[1]*1000,420,420,420,420]
      $ 929 "var_13≔get_actual_tcp_pose()"
      global var_13= get_actual_tcp_pose ()
      $ 930 "var_13≔p[var_13[0],var_13[1],0.1,var_13[3],var_13[4],var_13[5]]"
      global var_13=p[var_13[0],var_13[1],0.1,var_13[3],var_13[4],var_13[5]]
      $ 931 "Direction: Base Z+"
      global move_thread_flag_931=0
      thread move_thread_931():
        enter_critical
        move_thread_flag_931 = 1
        local towardsPos=calculate_point_to_move_towards(p[0.0,0.0,0.0,0.0,0.0,0.0], [0.0,0.0,1.0], 0.15)
        movel(towardsPos, a=0.03, v=0.015)
        move_thread_flag_931 = 2
        exit_critical
      end
      move_thread_flag_931 = 0
      move_thread_han_931 = run move_thread_931()
      while (True):
        sleep(1.0E-10)
        if (move_thread_flag_931 > 1):
          join move_thread_han_931
          $ 932 "Until (distance)"
          break
        end
        sync()
      end
      $ 933 "L1B1≔var_13"
      global L1B1=var_13
      $ 934 "Linea1_Buje2"
      $ 935 "Xfin≔((((L1B2x)*(-1)*Xp)-(Xd)-((L1B2y)*(1/m2)))*(-1))*(1)"
      global Xfin=((((L1B2x)*(-1)*Xp)-(Xd)-((L1B2y)*(1/m2)))*(-1))*(1)
      $ 936 "Yfin≔((((L1B2y)*(-1)*Yp)-(Yd)+((L1B2x)*(-1)*m1))*(-1))*(1)"
      global Yfin=((((L1B2y)*(-1)*Yp)-(Yd)+((L1B2x)*(-1)*m1))*(-1))*(1)
      $ 937 "rotaciones≔get_actual_tcp_pose()"
      global rotaciones= get_actual_tcp_pose ()
      $ 938 "var_3≔rotaciones[3]"
      global var_3=rotaciones[3]
      $ 939 "var_4≔rotaciones[4]"
      global var_4=rotaciones[4]
      $ 940 "var_5≔rotaciones[5]"
      global var_5=rotaciones[5]
      $ 941 "If broca≟1645"
      if (broca == 1645):
        $ 942 "PosFinal≔p[Xfin-0.00208915,Yfin-0.00208915,0.15,var_3,var_4,var_5]"
        global PosFinal=p[Xfin-0.00208915,Yfin-0.00208915,0.15,var_3,var_4,var_5]
      else:
        $ 943 "ElseIf broca≟1935"
        if (broca == 1935):
          $ 944 "PosFinal≔p[Xfin-0.00245745,Yfin-0.00245745,0.15,var_3,var_4,var_5]"
          global PosFinal=p[Xfin-0.00245745,Yfin-0.00245745,0.15,var_3,var_4,var_5]
        else:
          $ 945 "ElseIf broca≟217"
          if (broca == 217):
            $ 946 "PosFinal≔p[Xfin-0.0027559,Yfin-0.0027559,0.15,var_3,var_4,var_5]"
            global PosFinal=p[Xfin-0.0027559,Yfin-0.0027559,0.15,var_3,var_4,var_5]
          end
        end
      end
      $ 947 "Buje_Final≔PosFinal"
      global Buje_Final=PosFinal
      $ 948 "MoveJ"
      $ 949 "Buje_Final" "breakAfter"
      movej(Buje_Final, a=1.3962634015954636, v=1.0471975511965976)
      $ 950 "Wait: 1.0"
      sleep(1.0)
      $ 951 "Alturas"
      $ 952 "If P1h[2]<P2h[2]"
      if (P1h[2]<P2h[2]):
        $ 953 "tcp_chido≔get_actual_tcp_pose()"
        global tcp_chido= get_actual_tcp_pose ()
        $ 954 "offset_bajada≔p[tcp_chido[0],tcp_chido[1],((alta-0.0095)),tcp_chido[3],tcp_chido[4],tcp_chido[5]]"
        global offset_bajada=p[tcp_chido[0],tcp_chido[1],((alta-0.0095)),tcp_chido[3],tcp_chido[4],tcp_chido[5]]
        $ 955 "MoveL"
        $ 956 "offset_bajada" "breakAfter"
        movel(offset_bajada, a=0.03, v=0.015)
      else:
        $ 957 "Else" "noBreak"
        $ 958 "tcp_chido≔get_actual_tcp_pose()"
        global tcp_chido= get_actual_tcp_pose ()
        $ 959 "offset_bajada≔p[tcp_chido[0],tcp_chido[1],((alta-0.0095)-(altura/1000)),tcp_chido[3],tcp_chido[4],tcp_chido[5]]"
        global offset_bajada=p[tcp_chido[0],tcp_chido[1],((alta-0.0095)-(altura/1000)),tcp_chido[3],tcp_chido[4],tcp_chido[5]]
        $ 960 "MoveL"
        $ 961 "offset_bajada" "breakAfter"
        movel(offset_bajada, a=0.03, v=0.015)
      end
      $ 962 "MoveL"
      $ 963 "Freemove"
      $ 964 "Wait: 2.0"
      sleep(2.0)
      $ 965 "freedrive_mode()"
      freedrive_mode()
      $ 966 "Wait: 2.5"
      sleep(2.5)
      $ 967 "end_freedrive_mode()"
      end_freedrive_mode()
      $ 968 "var_13≔get_actual_tcp_pose()"
      global var_13= get_actual_tcp_pose ()
      $ 969 "var_13≔p[var_13[0]*1000,var_13[1]*1000,420,420,420,420]"
      global var_13=p[var_13[0]*1000,var_13[1]*1000,420,420,420,420]
      $ 970 "var_13≔get_actual_tcp_pose()"
      global var_13= get_actual_tcp_pose ()
      $ 971 "var_13≔p[var_13[0],var_13[1],0.1,var_13[3],var_13[4],var_13[5]]"
      global var_13=p[var_13[0],var_13[1],0.1,var_13[3],var_13[4],var_13[5]]
      $ 972 "Direction: Base Z+"
      global move_thread_flag_972=0
      thread move_thread_972():
        enter_critical
        move_thread_flag_972 = 1
        local towardsPos=calculate_point_to_move_towards(p[0.0,0.0,0.0,0.0,0.0,0.0], [0.0,0.0,1.0], 0.15)
        movel(towardsPos, a=0.03, v=0.015)
        move_thread_flag_972 = 2
        exit_critical
      end
      move_thread_flag_972 = 0
      move_thread_han_972 = run move_thread_972()
      while (True):
        sleep(1.0E-10)
        if (move_thread_flag_972 > 1):
          join move_thread_han_972
          $ 973 "Until (distance)"
          break
        end
        sync()
      end
      $ 974 "L1B2≔var_13"
      global L1B2=var_13
      $ 975 "Linea2_Buje2"
      $ 976 "Xfin≔((((L2B2x)*(-1)*Xp)-(Xd)-(L2B2y*(1/m2)))*(-1))*(1)"
      global Xfin=((((L2B2x)*(-1)*Xp)-(Xd)-(L2B2y*(1/m2)))*(-1))*(1)
      $ 977 "Yfin≔((((L2B2y)*(-1)*Yp)-(Yd)+((L2B2x)*(-1)*m1))*(-1))*(1)"
      global Yfin=((((L2B2y)*(-1)*Yp)-(Yd)+((L2B2x)*(-1)*m1))*(-1))*(1)
      $ 978 "rotaciones≔get_actual_tcp_pose()"
      global rotaciones= get_actual_tcp_pose ()
      $ 979 "var_3≔rotaciones[3]"
      global var_3=rotaciones[3]
      $ 980 "var_4≔rotaciones[4]"
      global var_4=rotaciones[4]
      $ 981 "var_5≔rotaciones[5]"
      global var_5=rotaciones[5]
      $ 982 "If broca≟1645"
      if (broca == 1645):
        $ 983 "PosFinal≔p[Xfin-0.00208915,Yfin-0.00208915,0.15,var_3,var_4,var_5]"
        global PosFinal=p[Xfin-0.00208915,Yfin-0.00208915,0.15,var_3,var_4,var_5]
      else:
        $ 984 "ElseIf broca≟1935"
        if (broca == 1935):
          $ 985 "PosFinal≔p[Xfin-0.00245745,Yfin-0.00245745,0.15,var_3,var_4,var_5]"
          global PosFinal=p[Xfin-0.00245745,Yfin-0.00245745,0.15,var_3,var_4,var_5]
        else:
          $ 986 "ElseIf broca≟217"
          if (broca == 217):
            $ 987 "PosFinal≔p[Xfin-0.0027559,Yfin-0.0027559,0.15,var_3,var_4,var_5]"
            global PosFinal=p[Xfin-0.0027559,Yfin-0.0027559,0.15,var_3,var_4,var_5]
          end
        end
      end
      $ 988 "Buje_Final≔PosFinal"
      global Buje_Final=PosFinal
      $ 989 "MoveJ"
      $ 990 "Buje_Final" "breakAfter"
      movej(Buje_Final, a=1.3962634015954636, v=1.0471975511965976)
      $ 991 "Wait: 1.0"
      sleep(1.0)
      $ 992 "Alturas"
      $ 993 "If P1h[2]<P2h[2]"
      if (P1h[2]<P2h[2]):
        $ 994 "tcp_chido≔get_actual_tcp_pose()"
        global tcp_chido= get_actual_tcp_pose ()
        $ 995 "offset_bajada≔p[tcp_chido[0],tcp_chido[1],((alta-0.0095)),tcp_chido[3],tcp_chido[4],tcp_chido[5]]"
        global offset_bajada=p[tcp_chido[0],tcp_chido[1],((alta-0.0095)),tcp_chido[3],tcp_chido[4],tcp_chido[5]]
        $ 996 "MoveL"
        $ 997 "offset_bajada" "breakAfter"
        movel(offset_bajada, a=0.03, v=0.015)
      else:
        $ 998 "Else" "noBreak"
        $ 999 "tcp_chido≔get_actual_tcp_pose()"
        global tcp_chido= get_actual_tcp_pose ()
        $ 1000 "offset_bajada≔p[tcp_chido[0],tcp_chido[1],((alta-0.0095)-(altura/1000)),tcp_chido[3],tcp_chido[4],tcp_chido[5]]"
        global offset_bajada=p[tcp_chido[0],tcp_chido[1],((alta-0.0095)-(altura/1000)),tcp_chido[3],tcp_chido[4],tcp_chido[5]]
        $ 1001 "MoveL"
        $ 1002 "offset_bajada" "breakAfter"
        movel(offset_bajada, a=0.03, v=0.015)
      end
      $ 1003 "MoveL"
      $ 1004 "Freemove"
      $ 1005 "Wait: 2.0"
      sleep(2.0)
      $ 1006 "freedrive_mode()"
      freedrive_mode()
      $ 1007 "Wait: 2.5"
      sleep(2.5)
      $ 1008 "end_freedrive_mode()"
      end_freedrive_mode()
      $ 1009 "var_13≔get_actual_tcp_pose()"
      global var_13= get_actual_tcp_pose ()
      $ 1010 "var_13≔p[var_13[0]*1000,var_13[1]*1000,420,420,420,420]"
      global var_13=p[var_13[0]*1000,var_13[1]*1000,420,420,420,420]
      $ 1011 "var_13≔get_actual_tcp_pose()"
      global var_13= get_actual_tcp_pose ()
      $ 1012 "var_13≔p[var_13[0],var_13[1],0.1,var_13[3],var_13[4],var_13[5]]"
      global var_13=p[var_13[0],var_13[1],0.1,var_13[3],var_13[4],var_13[5]]
      $ 1013 "Direction: Base Z+"
      global move_thread_flag_1013=0
      thread move_thread_1013():
        enter_critical
        move_thread_flag_1013 = 1
        local towardsPos=calculate_point_to_move_towards(p[0.0,0.0,0.0,0.0,0.0,0.0], [0.0,0.0,1.0], 0.15)
        movel(towardsPos, a=0.03, v=0.015)
        move_thread_flag_1013 = 2
        exit_critical
      end
      move_thread_flag_1013 = 0
      move_thread_han_1013 = run move_thread_1013()
      while (True):
        sleep(1.0E-10)
        if (move_thread_flag_1013 > 1):
          join move_thread_han_1013
          $ 1014 "Until (distance)"
          break
        end
        sync()
      end
      $ 1015 "L2B2≔var_13"
      global L2B2=var_13
      $ 1016 "Linea2_Buje1"
      $ 1017 "Xfin≔((((L2B1x)*(-1)*Xp)-(Xd)-((L2B1y)*(1/m2)))*(-1))*(1)"
      global Xfin=((((L2B1x)*(-1)*Xp)-(Xd)-((L2B1y)*(1/m2)))*(-1))*(1)
      $ 1018 "Yfin≔((((L2B1y)*(-1)*Yp)-(Yd)+((L2B1x)*(-1)*m1))*(-1))*(1)"
      global Yfin=((((L2B1y)*(-1)*Yp)-(Yd)+((L2B1x)*(-1)*m1))*(-1))*(1)
      $ 1019 "rotaciones≔get_actual_tcp_pose()"
      global rotaciones= get_actual_tcp_pose ()
      $ 1020 "var_3≔rotaciones[3]"
      global var_3=rotaciones[3]
      $ 1021 "var_4≔rotaciones[4]"
      global var_4=rotaciones[4]
      $ 1022 "var_5≔rotaciones[5]"
      global var_5=rotaciones[5]
      $ 1023 "If broca≟1645"
      if (broca == 1645):
        $ 1024 "PosFinal≔p[Xfin-0.00208915,Yfin-0.00208915,0.15,var_3,var_4,var_5]"
        global PosFinal=p[Xfin-0.00208915,Yfin-0.00208915,0.15,var_3,var_4,var_5]
      else:
        $ 1025 "ElseIf broca≟1935"
        if (broca == 1935):
          $ 1026 "PosFinal≔p[Xfin-0.00245745,Yfin-0.00245745,0.15,var_3,var_4,var_5]"
          global PosFinal=p[Xfin-0.00245745,Yfin-0.00245745,0.15,var_3,var_4,var_5]
        else:
          $ 1027 "ElseIf broca≟217"
          if (broca == 217):
            $ 1028 "PosFinal≔p[Xfin-0.0027559,Yfin-0.0027559,0.15,var_3,var_4,var_5]"
            global PosFinal=p[Xfin-0.0027559,Yfin-0.0027559,0.15,var_3,var_4,var_5]
          end
        end
      end
      $ 1029 "Buje_Final≔PosFinal"
      global Buje_Final=PosFinal
      $ 1030 "MoveJ"
      $ 1031 "Paso2_izq1" "breakAfter"
      movej(get_inverse_kin(Paso2_izq1_p, qnear=Paso2_izq1_q), a=1.3962634015954636, v=1.0471975511965976)
      $ 1032 "Buje_Final" "breakAfter"
      movej(Buje_Final, a=1.3962634015954636, v=1.0471975511965976)
      $ 1033 "Wait: 1.0"
      sleep(1.0)
      $ 1034 "Alturas"
      $ 1035 "If P1h[2]<P2h[2]"
      if (P1h[2]<P2h[2]):
        $ 1036 "tcp_chido≔get_actual_tcp_pose()"
        global tcp_chido= get_actual_tcp_pose ()
        $ 1037 "offset_bajada≔p[tcp_chido[0],tcp_chido[1],((alta-0.0095)-(altura/1000)),tcp_chido[3],tcp_chido[4],tcp_chido[5]]"
        global offset_bajada=p[tcp_chido[0],tcp_chido[1],((alta-0.0095)-(altura/1000)),tcp_chido[3],tcp_chido[4],tcp_chido[5]]
        $ 1038 "MoveL"
        $ 1039 "offset_bajada" "breakAfter"
        movel(offset_bajada, a=0.03, v=0.015)
      else:
        $ 1040 "Else" "noBreak"
        $ 1041 "tcp_chido≔get_actual_tcp_pose()"
        global tcp_chido= get_actual_tcp_pose ()
        $ 1042 "offset_bajada≔p[tcp_chido[0],tcp_chido[1],((alta-0.0095)),tcp_chido[3],tcp_chido[4],tcp_chido[5]]"
        global offset_bajada=p[tcp_chido[0],tcp_chido[1],((alta-0.0095)),tcp_chido[3],tcp_chido[4],tcp_chido[5]]
        $ 1043 "MoveL"
        $ 1044 "offset_bajada" "breakAfter"
        movel(offset_bajada, a=0.03, v=0.015)
      end
      $ 1045 "MoveL"
      $ 1046 "Freemove"
      $ 1047 "Wait: 2.0"
      sleep(2.0)
      $ 1048 "freedrive_mode()"
      freedrive_mode()
      $ 1049 "Wait: 2.5"
      sleep(2.5)
      $ 1050 "end_freedrive_mode()"
      end_freedrive_mode()
      $ 1051 "var_13≔get_actual_tcp_pose()"
      global var_13= get_actual_tcp_pose ()
      $ 1052 "var_13≔p[var_13[0]*1000,var_13[1]*1000,420,420,420,420]"
      global var_13=p[var_13[0]*1000,var_13[1]*1000,420,420,420,420]
      $ 1053 "var_13≔get_actual_tcp_pose()"
      global var_13= get_actual_tcp_pose ()
      $ 1054 "var_13≔p[var_13[0],var_13[1],0.1,var_13[3],var_13[4],var_13[5]]"
      global var_13=p[var_13[0],var_13[1],0.1,var_13[3],var_13[4],var_13[5]]
      $ 1055 "Direction: Base Z+"
      global move_thread_flag_1055=0
      thread move_thread_1055():
        enter_critical
        move_thread_flag_1055 = 1
        local towardsPos=calculate_point_to_move_towards(p[0.0,0.0,0.0,0.0,0.0,0.0], [0.0,0.0,1.0], 0.15)
        movel(towardsPos, a=0.03, v=0.015)
        move_thread_flag_1055 = 2
        exit_critical
      end
      move_thread_flag_1055 = 0
      move_thread_han_1055 = run move_thread_1055()
      while (True):
        sleep(1.0E-10)
        if (move_thread_flag_1055 > 1):
          join move_thread_han_1055
          $ 1056 "Until (distance)"
          break
        end
        sync()
      end
      $ 1057 "MoveJ"
      $ 1058 "Zona_izq1" "breakAfter"
      movej(get_inverse_kin(Zona_izq1_p, qnear=Zona_izq1_q), a=1.3962634015954636, v=1.0471975511965976)
      $ 1059 "L2B1≔var_13"
      global L2B1=var_13
      $ 1072 "Colocar broca"
      $ 1073 "Call Quitar_Broca_Chida"
      Quitar_Broca_Chida()
      $ 1074 "Call Poner_Broca"
      Poner_Broca()
      $ 1075 "Barrenado1"
      $ 1076 "Set mensaje_mw10=65"
      modbus_set_output_register("mensaje_mw10", 65)
      $ 1077 "Wait Continuar_M30=HI"
      while (modbus_get_signal_status("Continuar_M30") == False):
        sync()
      end
      $ 1078 "Wait: 1.0"
      sleep(1.0)
      $ 1079 "Set mensaje_mw10=150"
      modbus_set_output_register("mensaje_mw10", 150)
      $ 1080 "Wait: 1.0"
      sleep(1.0)
      $ 1081 "Linea 1 a 1645"
      $ 1082 "broca≔1645"
      global broca=1645
      $ 1083 "Buje_inicial"
      $ 1084 "Buje_Inicial≔L1B2"
      global Buje_Inicial=L1B2
      $ 1085 "Buje_final"
      $ 1086 "Buje_Final≔L1B1"
      global Buje_Final=L1B1
      $ 1087 "barrenosTotales≔27"
      global barrenosTotales=27
      $ 1088 "barrenoActual≔1"
      global barrenoActual=1
      $ 1089 "Loop barrenoActual≤barrenosTotales"
      while (barrenoActual <= barrenosTotales):
        $ 1090 "MoveL"
        $ 1091 "bajada_broca≔p[0,0,0.006,0,0,0]"
        global bajada_broca=p[0,0,0.006,0,0,0]
        $ 1092 "internos≔interpolate_pose(Buje_Inicial, Buje_Final, ((barrenoActual)-1)/((barrenosTotales)-1))"
        global internos= interpolate_pose (Buje_Inicial, Buje_Final, ((barrenoActual)-1)/((barrenosTotales)-1))
        $ 1093 "Alturas"
        $ 1094 "If barrenoActual≟3 or barrenoActual≟5 or barrenoActual≟7 or barrenoActual≟9 or barrenoActual≟11 or barrenoActual≟13 or barrenoActual≟15 or barrenoActual≟17 or barrenoActual≟19 or barrenoActual≟21 or barrenoActual≟23 or barrenoActual≟25 or barrenoActual≟27 or barrenoActual≟1"
        if (barrenoActual == 3  or  barrenoActual == 5  or  barrenoActual == 7  or  barrenoActual == 9  or  barrenoActual == 11  or  barrenoActual == 13  or  barrenoActual == 15  or  barrenoActual == 17  or  barrenoActual == 19  or  barrenoActual == 21  or  barrenoActual == 23  or  barrenoActual == 25  or  barrenoActual == 27  or  barrenoActual == 1):
          $ 1095 "Set mensaje_mw10=200"
          modbus_set_output_register("mensaje_mw10", 200)
          $ 1096 "Wait Continuar_M30=HI"
          while (modbus_get_signal_status("Continuar_M30") == False):
            sync()
          end
          $ 1097 "Wait: 1.0"
          sleep(1.0)
          $ 1098 "Set mensaje_mw10=150"
          modbus_set_output_register("mensaje_mw10", 150)
          $ 1099 "Wait: 1.0"
          sleep(1.0)
        end
        $ 1100 "MoveJ"
        $ 1101 "internos" "breakAfter"
        movej(internos, a=1.3962634015954636, v=1.0471975511965976)
        $ 1102 "Wait: 2.0"
        sleep(2.0)
        $ 1103 "If P1h[2]<P2h[2]"
        if (P1h[2]<P2h[2]):
          $ 1104 "acomodin≔(altura/(barrenosTotales-1))*(barrenoActual-1)"
          global acomodin=(altura/(barrenosTotales-1))*(barrenoActual-1)
          $ 1105 "tcp_chido≔get_actual_tcp_pose()"
          global tcp_chido= get_actual_tcp_pose ()
          $ 1106 "offset_bajada≔p[tcp_chido[0],tcp_chido[1],((alta-0.0095)-(acomodin/1000)),tcp_chido[3],tcp_chido[4],tcp_chido[5]]"
          global offset_bajada=p[tcp_chido[0],tcp_chido[1],((alta-0.0095)-(acomodin/1000)),tcp_chido[3],tcp_chido[4],tcp_chido[5]]
          $ 1107 "MoveL"
          $ 1108 "offset_bajada" "breakAfter"
          movel(offset_bajada, a=0.03, v=0.015)
        else:
          $ 1109 "Else" "noBreak"
          $ 1110 "acomodin≔(altura/(barrenosTotales-1))*(26-(barrenoActual-1))"
          global acomodin=(altura/(barrenosTotales-1))*(26-(barrenoActual-1))
          $ 1111 "tcp_chido≔get_actual_tcp_pose()"
          global tcp_chido= get_actual_tcp_pose ()
          $ 1112 "offset_bajada≔p[tcp_chido[0],tcp_chido[1],((alta-0.0095)-(acomodin/1000)),tcp_chido[3],tcp_chido[4],tcp_chido[5]]"
          global offset_bajada=p[tcp_chido[0],tcp_chido[1],((alta-0.0095)-(acomodin/1000)),tcp_chido[3],tcp_chido[4],tcp_chido[5]]
          $ 1113 "MoveL"
          $ 1114 "offset_bajada" "breakAfter"
          movel(offset_bajada, a=0.03, v=0.015)
        end
        $ 1115 "Freemove"
        $ 1116 "Wait: 2.0"
        sleep(2.0)
        $ 1117 "freedrive_mode()"
        freedrive_mode()
        $ 1118 "Wait: 2.5"
        sleep(2.5)
        $ 1119 "end_freedrive_mode()"
        end_freedrive_mode()
        $ 1120 "Wait: 0.3"
        sleep(0.3)
        $ 1121 "Set CO[1]=Encender"
        set_configurable_digital_out(1, True)
        $ 1122 "Wait: 1.0"
        sleep(1.0)
        $ 1123 "Wait: 0.3"
        sleep(0.3)
        $ 1124 "Wait: 0.3"
        sleep(0.3)
        $ 1125 "Wait: 0.3"
        sleep(0.3)
        $ 1126 "Loop 3 times"
        Loop_68 = 0
        while (Loop_68 < 3):
          $ 1127 "Poses_taladrado≔pose_sub(get_actual_tcp_pose(), bajada_broca)"
          global Poses_taladrado= pose_sub ( get_actual_tcp_pose (), bajada_broca)
          $ 1128 "Poses_taladrado" "breakAfter"
          movel(Poses_taladrado, a=0.005, v=0.001)
          $ 1129 "If bajada_broca≟p[0,0,0.018,0,0,0]"
          if (bajada_broca == p[0,0,0.018,0,0,0]):
            $ 1130 "num_barreno≔str_cat('Barreno: ',barrenoActual)"
            global num_barreno=str_cat("Barreno: ",barrenoActual)
            $ 1131 "tcp_actual≔get_actual_tcp_pose()"
            global tcp_actual= get_actual_tcp_pose ()
            $ 1132 "X_actual≔str_cat('     X: ',tcp_actual[0])"
            global X_actual=str_cat("     X: ",tcp_actual[0])
            $ 1133 "Y_actual≔str_cat('     Y: ',tcp_actual[1])"
            global Y_actual=str_cat("     Y: ",tcp_actual[1])
            $ 1134 "pos_barreno≔str_cat(X_actual,Y_actual)"
            global pos_barreno=str_cat(X_actual,Y_actual)
            $ 1135 "textmsg(num_barreno,pos_barreno)"
            textmsg(num_barreno,pos_barreno)
          end
          $ 1136 "Poses_taladrado≔pose_add(get_actual_tcp_pose(), bajada_broca)"
          global Poses_taladrado= pose_add ( get_actual_tcp_pose (), bajada_broca)
          $ 1137 "Poses_taladrado" "breakAfter"
          movel(Poses_taladrado, a=0.01, v=0.01)
          $ 1138 "bajada_broca≔pose_add(bajada_broca, p[0,0,0.006,0,0,0])"
          global bajada_broca= pose_add (bajada_broca, p[0,0,0.006,0,0,0])
          Loop_68 = Loop_68 + 1
        end
        $ 1139 "Direction: Base Z+"
        global move_thread_flag_1139=0
        thread move_thread_1139():
          enter_critical
          move_thread_flag_1139 = 1
          local towardsPos=calculate_point_to_move_towards(p[0.0,0.0,0.0,0.0,0.0,0.0], [0.0,0.0,1.0], 0.05)
          movel(towardsPos, a=0.04, v=0.03)
          move_thread_flag_1139 = 2
          exit_critical
        end
        move_thread_flag_1139 = 0
        move_thread_han_1139 = run move_thread_1139()
        while (True):
          sleep(1.0E-10)
          if (move_thread_flag_1139 > 1):
            join move_thread_han_1139
            $ 1140 "Until (distance)"
            break
          end
          sync()
        end
        $ 1141 "MoveJ"
        $ 1142 "internos" "breakAfter"
        movej(internos, a=1.3962634015954636, v=1.0471975511965976)
        $ 1143 "Wait: 0.3"
        sleep(0.3)
        $ 1144 "Set CO[1]=Apagar"
        set_configurable_digital_out(1, False)
        $ 1145 "Wait: 0.3"
        sleep(0.3)
        $ 1146 "If barrenoActual≟13 or barrenoActual≟27"
        if (barrenoActual == 13  or  barrenoActual == 27):
          $ 1147 "Direction: Base Z+"
          global move_thread_flag_1147=0
          thread move_thread_1147():
            enter_critical
            move_thread_flag_1147 = 1
            local towardsPos=calculate_point_to_move_towards(p[0.0,0.0,0.0,0.0,0.0,0.0], [0.0,0.0,1.0], 0.03)
            movel(towardsPos, a=0.04, v=0.03)
            move_thread_flag_1147 = 2
            exit_critical
          end
          move_thread_flag_1147 = 0
          move_thread_han_1147 = run move_thread_1147()
          while (True):
            sleep(1.0E-10)
            if (move_thread_flag_1147 > 1):
              join move_thread_han_1147
              $ 1148 "Until (distance)"
              break
            end
            sync()
          end
          $ 1149 "MoveJ"
          $ 1150 "Zona_izq1" "breakAfter"
          movej(get_inverse_kin(Zona_izq1_p, qnear=Zona_izq1_q), a=1.3962634015954636, v=1.0471975511965976)
          $ 1151 "Posicion_Cero" "breakAfter"
          movej(get_inverse_kin(Posicion_Cero_p, qnear=Posicion_Cero_q), a=1.3962634015954636, v=1.0471975511965976)
          $ 1152 "Call Quitar_Broca_Chida"
          Quitar_Broca_Chida()
          $ 1153 "Call Poner_Broca"
          Poner_Broca()
          $ 1154 "MoveJ"
          $ 1155 "Posicion_Cero" "breakAfter"
          movej(get_inverse_kin(Posicion_Cero_p, qnear=Posicion_Cero_q), a=1.3962634015954636, v=1.0471975511965976)
          $ 1156 "Zona_izq1" "breakAfter"
          movej(get_inverse_kin(Zona_izq1_p, qnear=Zona_izq1_q), a=1.3962634015954636, v=1.0471975511965976)
        end
        $ 1157 "barrenoActual≔barrenoActual+1"
        global barrenoActual=barrenoActual+1
      end
      $ 1158 "Linea 2 a 1645"
      $ 1159 "broca≔1645"
      global broca=1645
      $ 1160 "Buje_inicial"
      $ 1161 "Buje_Inicial≔L2B2"
      global Buje_Inicial=L2B2
      $ 1162 "Buje_final"
      $ 1163 "Buje_Final≔L2B1"
      global Buje_Final=L2B1
      $ 1164 "barrenosTotales≔27"
      global barrenosTotales=27
      $ 1165 "barrenoActual≔1"
      global barrenoActual=1
      $ 1166 "Loop barrenoActual≤barrenosTotales"
      while (barrenoActual <= barrenosTotales):
        $ 1167 "MoveL"
        $ 1168 "bajada_broca≔p[0,0,0.006,0,0,0]"
        global bajada_broca=p[0,0,0.006,0,0,0]
        $ 1169 "internos≔interpolate_pose(Buje_Inicial, Buje_Final, ((barrenoActual)-1)/((barrenosTotales)-1))"
        global internos= interpolate_pose (Buje_Inicial, Buje_Final, ((barrenoActual)-1)/((barrenosTotales)-1))
        $ 1170 "Alturas"
        $ 1171 "If barrenoActual≟3 or barrenoActual≟5 or barrenoActual≟7 or barrenoActual≟9 or barrenoActual≟11 or barrenoActual≟13 or barrenoActual≟15 or barrenoActual≟17 or barrenoActual≟19 or barrenoActual≟21 or barrenoActual≟23 or barrenoActual≟25 or barrenoActual≟27 or barrenoActual≟1"
        if (barrenoActual == 3  or  barrenoActual == 5  or  barrenoActual == 7  or  barrenoActual == 9  or  barrenoActual == 11  or  barrenoActual == 13  or  barrenoActual == 15  or  barrenoActual == 17  or  barrenoActual == 19  or  barrenoActual == 21  or  barrenoActual == 23  or  barrenoActual == 25  or  barrenoActual == 27  or  barrenoActual == 1):
          $ 1172 "Set mensaje_mw10=200"
          modbus_set_output_register("mensaje_mw10", 200)
          $ 1173 "Wait Continuar_M30=HI"
          while (modbus_get_signal_status("Continuar_M30") == False):
            sync()
          end
          $ 1174 "Wait: 1.0"
          sleep(1.0)
          $ 1175 "Set mensaje_mw10=150"
          modbus_set_output_register("mensaje_mw10", 150)
          $ 1176 "Wait: 1.0"
          sleep(1.0)
        end
        $ 1177 "MoveJ"
        $ 1178 "internos" "breakAfter"
        movej(internos, a=1.3962634015954636, v=1.0471975511965976)
        $ 1179 "Wait: 2.0"
        sleep(2.0)
        $ 1180 "If P1h[2]<P2h[2]"
        if (P1h[2]<P2h[2]):
          $ 1181 "acomodin≔(altura/(barrenosTotales-1))*(barrenoActual-1)"
          global acomodin=(altura/(barrenosTotales-1))*(barrenoActual-1)
          $ 1182 "tcp_chido≔get_actual_tcp_pose()"
          global tcp_chido= get_actual_tcp_pose ()
          $ 1183 "offset_bajada≔p[tcp_chido[0],tcp_chido[1],((alta-0.0095)-(acomodin/1000)),tcp_chido[3],tcp_chido[4],tcp_chido[5]]"
          global offset_bajada=p[tcp_chido[0],tcp_chido[1],((alta-0.0095)-(acomodin/1000)),tcp_chido[3],tcp_chido[4],tcp_chido[5]]
          $ 1184 "MoveL"
          $ 1185 "offset_bajada" "breakAfter"
          movel(offset_bajada, a=0.03, v=0.015)
        else:
          $ 1186 "Else" "noBreak"
          $ 1187 "acomodin≔(altura/(barrenosTotales-1))*(26-(barrenoActual-1))"
          global acomodin=(altura/(barrenosTotales-1))*(26-(barrenoActual-1))
          $ 1188 "tcp_chido≔get_actual_tcp_pose()"
          global tcp_chido= get_actual_tcp_pose ()
          $ 1189 "offset_bajada≔p[tcp_chido[0],tcp_chido[1],((alta-0.0095)-(acomodin/1000)),tcp_chido[3],tcp_chido[4],tcp_chido[5]]"
          global offset_bajada=p[tcp_chido[0],tcp_chido[1],((alta-0.0095)-(acomodin/1000)),tcp_chido[3],tcp_chido[4],tcp_chido[5]]
          $ 1190 "MoveL"
          $ 1191 "offset_bajada" "breakAfter"
          movel(offset_bajada, a=0.03, v=0.015)
        end
        $ 1192 "Freemove"
        $ 1193 "Wait: 2.0"
        sleep(2.0)
        $ 1194 "freedrive_mode()"
        freedrive_mode()
        $ 1195 "Wait: 2.5"
        sleep(2.5)
        $ 1196 "end_freedrive_mode()"
        end_freedrive_mode()
        $ 1197 "Wait: 0.3"
        sleep(0.3)
        $ 1198 "Set CO[1]=Encender"
        set_configurable_digital_out(1, True)
        $ 1199 "Wait: 1.0"
        sleep(1.0)
        $ 1200 "Wait: 0.3"
        sleep(0.3)
        $ 1201 "Wait: 0.3"
        sleep(0.3)
        $ 1202 "Wait: 0.3"
        sleep(0.3)
        $ 1203 "Loop 3 times"
        Loop_70 = 0
        while (Loop_70 < 3):
          $ 1204 "Poses_taladrado≔pose_sub(get_actual_tcp_pose(), bajada_broca)"
          global Poses_taladrado= pose_sub ( get_actual_tcp_pose (), bajada_broca)
          $ 1205 "Poses_taladrado" "breakAfter"
          movel(Poses_taladrado, a=0.005, v=0.001)
          $ 1206 "If bajada_broca≟p[0,0,0.018,0,0,0]"
          if (bajada_broca == p[0,0,0.018,0,0,0]):
            $ 1207 "num_barreno≔str_cat('Barreno: ',barrenoActual)"
            global num_barreno=str_cat("Barreno: ",barrenoActual)
            $ 1208 "tcp_actual≔get_actual_tcp_pose()"
            global tcp_actual= get_actual_tcp_pose ()
            $ 1209 "X_actual≔str_cat('     X: ',tcp_actual[0])"
            global X_actual=str_cat("     X: ",tcp_actual[0])
            $ 1210 "Y_actual≔str_cat('     Y: ',tcp_actual[1])"
            global Y_actual=str_cat("     Y: ",tcp_actual[1])
            $ 1211 "pos_barreno≔str_cat(X_actual,Y_actual)"
            global pos_barreno=str_cat(X_actual,Y_actual)
            $ 1212 "textmsg(num_barreno,pos_barreno)"
            textmsg(num_barreno,pos_barreno)
          end
          $ 1213 "Poses_taladrado≔pose_add(get_actual_tcp_pose(), bajada_broca)"
          global Poses_taladrado= pose_add ( get_actual_tcp_pose (), bajada_broca)
          $ 1214 "Poses_taladrado" "breakAfter"
          movel(Poses_taladrado, a=0.01, v=0.01)
          $ 1215 "bajada_broca≔pose_add(bajada_broca, p[0,0,0.006,0,0,0])"
          global bajada_broca= pose_add (bajada_broca, p[0,0,0.006,0,0,0])
          Loop_70 = Loop_70 + 1
        end
        $ 1216 "Direction: Base Z+"
        global move_thread_flag_1216=0
        thread move_thread_1216():
          enter_critical
          move_thread_flag_1216 = 1
          local towardsPos=calculate_point_to_move_towards(p[0.0,0.0,0.0,0.0,0.0,0.0], [0.0,0.0,1.0], 0.05)
          movel(towardsPos, a=0.04, v=0.03)
          move_thread_flag_1216 = 2
          exit_critical
        end
        move_thread_flag_1216 = 0
        move_thread_han_1216 = run move_thread_1216()
        while (True):
          sleep(1.0E-10)
          if (move_thread_flag_1216 > 1):
            join move_thread_han_1216
            $ 1217 "Until (distance)"
            break
          end
          sync()
        end
        $ 1218 "MoveJ"
        $ 1219 "internos" "breakAfter"
        movej(internos, a=1.3962634015954636, v=1.0471975511965976)
        $ 1220 "Wait: 0.3"
        sleep(0.3)
        $ 1221 "Set CO[1]=Apagar"
        set_configurable_digital_out(1, False)
        $ 1222 "Wait: 0.3"
        sleep(0.3)
        $ 1223 "If barrenoActual≟13"
        if (barrenoActual == 13):
          $ 1224 "Direction: Base Z+"
          global move_thread_flag_1224=0
          thread move_thread_1224():
            enter_critical
            move_thread_flag_1224 = 1
            local towardsPos=calculate_point_to_move_towards(p[0.0,0.0,0.0,0.0,0.0,0.0], [0.0,0.0,1.0], 0.03)
            movel(towardsPos, a=1.2, v=0.25)
            move_thread_flag_1224 = 2
            exit_critical
          end
          move_thread_flag_1224 = 0
          move_thread_han_1224 = run move_thread_1224()
          while (True):
            sleep(1.0E-10)
            if (move_thread_flag_1224 > 1):
              join move_thread_han_1224
              $ 1225 "Until (distance)"
              break
            end
            sync()
          end
          $ 1226 "MoveJ"
          $ 1227 "Zona_izq1" "breakAfter"
          movej(get_inverse_kin(Zona_izq1_p, qnear=Zona_izq1_q), a=1.3962634015954636, v=1.0471975511965976)
          $ 1228 "Posicion_Cero" "breakAfter"
          movej(get_inverse_kin(Posicion_Cero_p, qnear=Posicion_Cero_q), a=1.3962634015954636, v=1.0471975511965976)
          $ 1229 "Call Quitar_Broca_Chida"
          Quitar_Broca_Chida()
          $ 1230 "Call Poner_Broca"
          Poner_Broca()
          $ 1231 "MoveJ"
          $ 1232 "Posicion_Cero" "breakAfter"
          movej(get_inverse_kin(Posicion_Cero_p, qnear=Posicion_Cero_q), a=1.3962634015954636, v=1.0471975511965976)
          $ 1233 "Zona_izq1" "breakAfter"
          movej(get_inverse_kin(Zona_izq1_p, qnear=Zona_izq1_q), a=1.3962634015954636, v=1.0471975511965976)
        else:
          $ 1234 "ElseIf barrenoActual≟27"
          if (barrenoActual == 27):
            $ 1235 "Direction: Base Z+"
            global move_thread_flag_1235=0
            thread move_thread_1235():
              enter_critical
              move_thread_flag_1235 = 1
              local towardsPos=calculate_point_to_move_towards(p[0.0,0.0,0.0,0.0,0.0,0.0], [0.0,0.0,1.0], 0.03)
              movel(towardsPos, a=1.2, v=0.25)
              move_thread_flag_1235 = 2
              exit_critical
            end
            move_thread_flag_1235 = 0
            move_thread_han_1235 = run move_thread_1235()
            while (True):
              sleep(1.0E-10)
              if (move_thread_flag_1235 > 1):
                join move_thread_han_1235
                $ 1236 "Until (distance)"
                break
              end
              sync()
            end
            $ 1237 "MoveJ"
            $ 1238 "Zona_izq1" "breakAfter"
            movej(get_inverse_kin(Zona_izq1_p, qnear=Zona_izq1_q), a=1.3962634015954636, v=1.0471975511965976)
            $ 1239 "Posicion_Cero" "breakAfter"
            movej(get_inverse_kin(Posicion_Cero_p, qnear=Posicion_Cero_q), a=1.3962634015954636, v=1.0471975511965976)
            $ 1240 "Call Quitar_Broca_Chida"
            Quitar_Broca_Chida()
            $ 1241 "Set carrusel_home=Encender"
            modbus_set_output_signal("carrusel_home", True)
            $ 1242 "Wait: 1.0"
            sleep(1.0)
            $ 1243 "Set carrusel_home=Apagar"
            modbus_set_output_signal("carrusel_home", False)
            $ 1244 "Set mensaje_mw10=70"
            modbus_set_output_register("mensaje_mw10", 70)
            $ 1245 "Wait Continuar_M30=HI"
            while (modbus_get_signal_status("Continuar_M30") == False):
              sync()
            end
            $ 1246 "Wait: 1.0"
            sleep(1.0)
            $ 1247 "Set mensaje_mw10=120"
            modbus_set_output_register("mensaje_mw10", 120)
            $ 1248 "Wait Continuar_M30=HI"
            while (modbus_get_signal_status("Continuar_M30") == False):
              sync()
            end
            $ 1249 "Wait: 1.0"
            sleep(1.0)
            $ 1250 "Set carrusel_home=Encender"
            modbus_set_output_signal("carrusel_home", True)
            $ 1251 "Wait: 1.0"
            sleep(1.0)
            $ 1252 "Set carrusel_home=Apagar"
            modbus_set_output_signal("carrusel_home", False)
            $ 1253 "Set mensaje_mw10=75"
            modbus_set_output_register("mensaje_mw10", 75)
            $ 1254 "Wait Continuar_M30=HI"
            while (modbus_get_signal_status("Continuar_M30") == False):
              sync()
            end
            $ 1255 "Wait: 1.0"
            sleep(1.0)
            $ 1256 "Call Poner_Broca"
            Poner_Broca()
            $ 1257 "broca≔1935"
            global broca=1935
            $ 1258 "MoveJ"
            $ 1259 "Posicion_Cero" "breakAfter"
            movej(get_inverse_kin(Posicion_Cero_p, qnear=Posicion_Cero_q), a=1.3962634015954636, v=1.0471975511965976)
            $ 1260 "Zona_izq1" "breakAfter"
            movej(get_inverse_kin(Zona_izq1_p, qnear=Zona_izq1_q), a=1.3962634015954636, v=1.0471975511965976)
            $ 1261 "Set mensaje_mw10=80"
            modbus_set_output_register("mensaje_mw10", 80)
            $ 1262 "Wait Continuar_M30=HI"
            while (modbus_get_signal_status("Continuar_M30") == False):
              sync()
            end
            $ 1263 "Wait: 1.0"
            sleep(1.0)
            $ 1264 "Set mensaje_mw10=150"
            modbus_set_output_register("mensaje_mw10", 150)
            $ 1265 "Wait Continuar_M30=HI"
            while (modbus_get_signal_status("Continuar_M30") == False):
              sync()
            end
            $ 1266 "Wait: 1.0"
            sleep(1.0)
          end
        end
        $ 1267 "barrenoActual≔barrenoActual+1"
        global barrenoActual=barrenoActual+1
      end
      $ 1268 "Linea 1 a 1935"
      $ 1269 "broca≔1935"
      global broca=1935
      $ 1270 "Buje_inicial"
      $ 1271 "Buje_Inicial≔L1B2"
      global Buje_Inicial=L1B2
      $ 1272 "Buje_final"
      $ 1273 "Buje_Final≔L1B1"
      global Buje_Final=L1B1
      $ 1274 "barrenosTotales≔27"
      global barrenosTotales=27
      $ 1275 "barrenoActual≔1"
      global barrenoActual=1
      $ 1276 "Loop barrenoActual≤barrenosTotales"
      while (barrenoActual <= barrenosTotales):
        $ 1277 "MoveL"
        $ 1278 "bajada_broca≔p[0,0,0.009,0,0,0]"
        global bajada_broca=p[0,0,0.009,0,0,0]
        $ 1279 "internos≔interpolate_pose(Buje_Inicial, Buje_Final, ((barrenoActual)-1)/((barrenosTotales)-1))"
        global internos= interpolate_pose (Buje_Inicial, Buje_Final, ((barrenoActual)-1)/((barrenosTotales)-1))
        $ 1280 "Alturas"
        $ 1281 "If barrenoActual≟3 or barrenoActual≟5 or barrenoActual≟7 or barrenoActual≟9 or barrenoActual≟11 or barrenoActual≟13 or barrenoActual≟15 or barrenoActual≟17 or barrenoActual≟19 or barrenoActual≟21 or barrenoActual≟23 or barrenoActual≟25 or barrenoActual≟27 or barrenoActual≟1"
        if (barrenoActual == 3  or  barrenoActual == 5  or  barrenoActual == 7  or  barrenoActual == 9  or  barrenoActual == 11  or  barrenoActual == 13  or  barrenoActual == 15  or  barrenoActual == 17  or  barrenoActual == 19  or  barrenoActual == 21  or  barrenoActual == 23  or  barrenoActual == 25  or  barrenoActual == 27  or  barrenoActual == 1):
          $ 1282 "Set mensaje_mw10=200"
          modbus_set_output_register("mensaje_mw10", 200)
          $ 1283 "Wait Continuar_M30=HI"
          while (modbus_get_signal_status("Continuar_M30") == False):
            sync()
          end
          $ 1284 "Wait: 1.0"
          sleep(1.0)
          $ 1285 "Set mensaje_mw10=150"
          modbus_set_output_register("mensaje_mw10", 150)
          $ 1286 "Wait: 1.0"
          sleep(1.0)
        end
        $ 1287 "MoveJ"
        $ 1288 "internos" "breakAfter"
        movej(internos, a=1.3962634015954636, v=1.0471975511965976)
        $ 1289 "Wait: 2.0"
        sleep(2.0)
        $ 1290 "If P1h[2]<P2h[2]"
        if (P1h[2]<P2h[2]):
          $ 1291 "acomodin≔(altura/(barrenosTotales-1))*(barrenoActual-1)"
          global acomodin=(altura/(barrenosTotales-1))*(barrenoActual-1)
          $ 1292 "tcp_chido≔get_actual_tcp_pose()"
          global tcp_chido= get_actual_tcp_pose ()
          $ 1293 "offset_bajada≔p[tcp_chido[0],tcp_chido[1],((alta-0.0095)-(acomodin/1000)),tcp_chido[3],tcp_chido[4],tcp_chido[5]]"
          global offset_bajada=p[tcp_chido[0],tcp_chido[1],((alta-0.0095)-(acomodin/1000)),tcp_chido[3],tcp_chido[4],tcp_chido[5]]
          $ 1294 "MoveL"
          $ 1295 "offset_bajada" "breakAfter"
          movel(offset_bajada, a=0.03, v=0.015)
        else:
          $ 1296 "Else" "noBreak"
          $ 1297 "acomodin≔(altura/(barrenosTotales-1))*(26-(barrenoActual-1))"
          global acomodin=(altura/(barrenosTotales-1))*(26-(barrenoActual-1))
          $ 1298 "tcp_chido≔get_actual_tcp_pose()"
          global tcp_chido= get_actual_tcp_pose ()
          $ 1299 "offset_bajada≔p[tcp_chido[0],tcp_chido[1],((alta-0.0095)-(acomodin/1000)),tcp_chido[3],tcp_chido[4],tcp_chido[5]]"
          global offset_bajada=p[tcp_chido[0],tcp_chido[1],((alta-0.0095)-(acomodin/1000)),tcp_chido[3],tcp_chido[4],tcp_chido[5]]
          $ 1300 "MoveL"
          $ 1301 "offset_bajada" "breakAfter"
          movel(offset_bajada, a=0.03, v=0.015)
        end
        $ 1302 "Freemove"
        $ 1303 "Wait: 2.0"
        sleep(2.0)
        $ 1304 "freedrive_mode()"
        freedrive_mode()
        $ 1305 "Wait: 2.5"
        sleep(2.5)
        $ 1306 "end_freedrive_mode()"
        end_freedrive_mode()
        $ 1307 "Wait: 0.3"
        sleep(0.3)
        $ 1308 "Set CO[1]=Encender"
        set_configurable_digital_out(1, True)
        $ 1309 "Wait: 1.0"
        sleep(1.0)
        $ 1310 "Wait: 0.3"
        sleep(0.3)
        $ 1311 "Wait: 0.3"
        sleep(0.3)
        $ 1312 "Wait: 0.3"
        sleep(0.3)
        $ 1313 "Loop 2 times"
        Loop_72 = 0
        while (Loop_72 < 2):
          $ 1314 "Poses_taladrado≔pose_sub(get_actual_tcp_pose(), bajada_broca)"
          global Poses_taladrado= pose_sub ( get_actual_tcp_pose (), bajada_broca)
          $ 1315 "Poses_taladrado" "breakAfter"
          movel(Poses_taladrado, a=0.005, v=0.001)
          $ 1316 "If bajada_broca≟p[0,0,0.018,0,0,0]"
          if (bajada_broca == p[0,0,0.018,0,0,0]):
            $ 1317 "num_barreno≔str_cat('Barreno: ',barrenoActual)"
            global num_barreno=str_cat("Barreno: ",barrenoActual)
            $ 1318 "tcp_actual≔get_actual_tcp_pose()"
            global tcp_actual= get_actual_tcp_pose ()
            $ 1319 "X_actual≔str_cat('     X: ',tcp_actual[0])"
            global X_actual=str_cat("     X: ",tcp_actual[0])
            $ 1320 "Y_actual≔str_cat('     Y: ',tcp_actual[1])"
            global Y_actual=str_cat("     Y: ",tcp_actual[1])
            $ 1321 "pos_barreno≔str_cat(X_actual,Y_actual)"
            global pos_barreno=str_cat(X_actual,Y_actual)
            $ 1322 "textmsg(num_barreno,pos_barreno)"
            textmsg(num_barreno,pos_barreno)
          end
          $ 1323 "Poses_taladrado≔pose_add(get_actual_tcp_pose(), bajada_broca)"
          global Poses_taladrado= pose_add ( get_actual_tcp_pose (), bajada_broca)
          $ 1324 "Poses_taladrado" "breakAfter"
          movel(Poses_taladrado, a=0.01, v=0.01)
          $ 1325 "bajada_broca≔pose_add(bajada_broca, p[0,0,0.009,0,0,0])"
          global bajada_broca= pose_add (bajada_broca, p[0,0,0.009,0,0,0])
          Loop_72 = Loop_72 + 1
        end
        $ 1326 "Direction: Base Z+"
        global move_thread_flag_1326=0
        thread move_thread_1326():
          enter_critical
          move_thread_flag_1326 = 1
          local towardsPos=calculate_point_to_move_towards(p[0.0,0.0,0.0,0.0,0.0,0.0], [0.0,0.0,1.0], 0.05)
          movel(towardsPos, a=0.04, v=0.03)
          move_thread_flag_1326 = 2
          exit_critical
        end
        move_thread_flag_1326 = 0
        move_thread_han_1326 = run move_thread_1326()
        while (True):
          sleep(1.0E-10)
          if (move_thread_flag_1326 > 1):
            join move_thread_han_1326
            $ 1327 "Until (distance)"
            break
          end
          sync()
        end
        $ 1328 "MoveJ"
        $ 1329 "internos" "breakAfter"
        movej(internos, a=1.3962634015954636, v=1.0471975511965976)
        $ 1330 "Wait: 0.3"
        sleep(0.3)
        $ 1331 "Set CO[1]=Apagar"
        set_configurable_digital_out(1, False)
        $ 1332 "Wait: 0.3"
        sleep(0.3)
        $ 1333 "If barrenoActual≟13 or barrenoActual≟27"
        if (barrenoActual == 13  or  barrenoActual == 27):
          $ 1334 "Direction: Base Z+"
          global move_thread_flag_1334=0
          thread move_thread_1334():
            enter_critical
            move_thread_flag_1334 = 1
            local towardsPos=calculate_point_to_move_towards(p[0.0,0.0,0.0,0.0,0.0,0.0], [0.0,0.0,1.0], 0.03)
            movel(towardsPos, a=1.2, v=0.25)
            move_thread_flag_1334 = 2
            exit_critical
          end
          move_thread_flag_1334 = 0
          move_thread_han_1334 = run move_thread_1334()
          while (True):
            sleep(1.0E-10)
            if (move_thread_flag_1334 > 1):
              join move_thread_han_1334
              $ 1335 "Until (distance)"
              break
            end
            sync()
          end
          $ 1336 "MoveJ"
          $ 1337 "Zona_izq1" "breakAfter"
          movej(get_inverse_kin(Zona_izq1_p, qnear=Zona_izq1_q), a=1.3962634015954636, v=1.0471975511965976)
          $ 1338 "Posicion_Cero" "breakAfter"
          movej(get_inverse_kin(Posicion_Cero_p, qnear=Posicion_Cero_q), a=1.3962634015954636, v=1.0471975511965976)
          $ 1339 "Call Quitar_Broca_Chida"
          Quitar_Broca_Chida()
          $ 1340 "Call Poner_Broca"
          Poner_Broca()
          $ 1341 "MoveJ"
          $ 1342 "Posicion_Cero" "breakAfter"
          movej(get_inverse_kin(Posicion_Cero_p, qnear=Posicion_Cero_q), a=1.3962634015954636, v=1.0471975511965976)
          $ 1343 "Zona_izq1" "breakAfter"
          movej(get_inverse_kin(Zona_izq1_p, qnear=Zona_izq1_q), a=1.3962634015954636, v=1.0471975511965976)
        end
        $ 1344 "barrenoActual≔barrenoActual+1"
        global barrenoActual=barrenoActual+1
      end
      $ 1345 "Linea 2 a 1935"
      $ 1346 "broca≔1935"
      global broca=1935
      $ 1347 "Buje_inicial"
      $ 1348 "Buje_Inicial≔L2B2"
      global Buje_Inicial=L2B2
      $ 1349 "Buje_final"
      $ 1350 "Buje_Final≔L2B1"
      global Buje_Final=L2B1
      $ 1351 "barrenosTotales≔27"
      global barrenosTotales=27
      $ 1352 "barrenoActual≔1"
      global barrenoActual=1
      $ 1353 "Loop barrenoActual≤barrenosTotales"
      while (barrenoActual <= barrenosTotales):
        $ 1354 "MoveL"
        $ 1355 "bajada_broca≔p[0,0,0.009,0,0,0]"
        global bajada_broca=p[0,0,0.009,0,0,0]
        $ 1356 "internos≔interpolate_pose(Buje_Inicial, Buje_Final, ((barrenoActual)-1)/((barrenosTotales)-1))"
        global internos= interpolate_pose (Buje_Inicial, Buje_Final, ((barrenoActual)-1)/((barrenosTotales)-1))
        $ 1357 "Alturas"
        $ 1358 "If barrenoActual≟3 or barrenoActual≟5 or barrenoActual≟7 or barrenoActual≟9 or barrenoActual≟11 or barrenoActual≟13 or barrenoActual≟15 or barrenoActual≟17 or barrenoActual≟19 or barrenoActual≟21 or barrenoActual≟23 or barrenoActual≟25 or barrenoActual≟27 or barrenoActual≟1"
        if (barrenoActual == 3  or  barrenoActual == 5  or  barrenoActual == 7  or  barrenoActual == 9  or  barrenoActual == 11  or  barrenoActual == 13  or  barrenoActual == 15  or  barrenoActual == 17  or  barrenoActual == 19  or  barrenoActual == 21  or  barrenoActual == 23  or  barrenoActual == 25  or  barrenoActual == 27  or  barrenoActual == 1):
          $ 1359 "Set mensaje_mw10=200"
          modbus_set_output_register("mensaje_mw10", 200)
          $ 1360 "Wait Continuar_M30=HI"
          while (modbus_get_signal_status("Continuar_M30") == False):
            sync()
          end
          $ 1361 "Wait: 1.0"
          sleep(1.0)
          $ 1362 "Set mensaje_mw10=150"
          modbus_set_output_register("mensaje_mw10", 150)
          $ 1363 "Wait: 1.0"
          sleep(1.0)
        end
        $ 1364 "MoveJ"
        $ 1365 "internos" "breakAfter"
        movej(internos, a=1.3962634015954636, v=1.0471975511965976)
        $ 1366 "Wait: 2.0"
        sleep(2.0)
        $ 1367 "If P1h[2]<P2h[2]"
        if (P1h[2]<P2h[2]):
          $ 1368 "acomodin≔(altura/(barrenosTotales-1))*(barrenoActual-1)"
          global acomodin=(altura/(barrenosTotales-1))*(barrenoActual-1)
          $ 1369 "tcp_chido≔get_actual_tcp_pose()"
          global tcp_chido= get_actual_tcp_pose ()
          $ 1370 "offset_bajada≔p[tcp_chido[0],tcp_chido[1],((alta-0.0095)-(acomodin/1000)),tcp_chido[3],tcp_chido[4],tcp_chido[5]]"
          global offset_bajada=p[tcp_chido[0],tcp_chido[1],((alta-0.0095)-(acomodin/1000)),tcp_chido[3],tcp_chido[4],tcp_chido[5]]
          $ 1371 "MoveL"
          $ 1372 "offset_bajada" "breakAfter"
          movel(offset_bajada, a=0.03, v=0.015)
        else:
          $ 1373 "Else" "noBreak"
          $ 1374 "acomodin≔(altura/(barrenosTotales-1))*(26-(barrenoActual-1))"
          global acomodin=(altura/(barrenosTotales-1))*(26-(barrenoActual-1))
          $ 1375 "tcp_chido≔get_actual_tcp_pose()"
          global tcp_chido= get_actual_tcp_pose ()
          $ 1376 "offset_bajada≔p[tcp_chido[0],tcp_chido[1],((alta-0.0095)-(acomodin/1000)),tcp_chido[3],tcp_chido[4],tcp_chido[5]]"
          global offset_bajada=p[tcp_chido[0],tcp_chido[1],((alta-0.0095)-(acomodin/1000)),tcp_chido[3],tcp_chido[4],tcp_chido[5]]
          $ 1377 "MoveL"
          $ 1378 "offset_bajada" "breakAfter"
          movel(offset_bajada, a=0.03, v=0.015)
        end
        $ 1379 "Freemove"
        $ 1380 "Wait: 2.0"
        sleep(2.0)
        $ 1381 "freedrive_mode()"
        freedrive_mode()
        $ 1382 "Wait: 2.5"
        sleep(2.5)
        $ 1383 "end_freedrive_mode()"
        end_freedrive_mode()
        $ 1384 "Wait: 0.3"
        sleep(0.3)
        $ 1385 "Set CO[1]=Encender"
        set_configurable_digital_out(1, True)
        $ 1386 "Wait: 1.0"
        sleep(1.0)
        $ 1387 "Wait: 0.3"
        sleep(0.3)
        $ 1388 "Wait: 0.3"
        sleep(0.3)
        $ 1389 "Wait: 0.3"
        sleep(0.3)
        $ 1390 "Loop 2 times"
        Loop_74 = 0
        while (Loop_74 < 2):
          $ 1391 "Poses_taladrado≔pose_sub(get_actual_tcp_pose(), bajada_broca)"
          global Poses_taladrado= pose_sub ( get_actual_tcp_pose (), bajada_broca)
          $ 1392 "Poses_taladrado" "breakAfter"
          movel(Poses_taladrado, a=0.005, v=0.001)
          $ 1393 "If bajada_broca≟p[0,0,0.018,0,0,0]"
          if (bajada_broca == p[0,0,0.018,0,0,0]):
            $ 1394 "num_barreno≔str_cat('Barreno: ',barrenoActual)"
            global num_barreno=str_cat("Barreno: ",barrenoActual)
            $ 1395 "tcp_actual≔get_actual_tcp_pose()"
            global tcp_actual= get_actual_tcp_pose ()
            $ 1396 "X_actual≔str_cat('     X: ',tcp_actual[0])"
            global X_actual=str_cat("     X: ",tcp_actual[0])
            $ 1397 "Y_actual≔str_cat('     Y: ',tcp_actual[1])"
            global Y_actual=str_cat("     Y: ",tcp_actual[1])
            $ 1398 "pos_barreno≔str_cat(X_actual,Y_actual)"
            global pos_barreno=str_cat(X_actual,Y_actual)
            $ 1399 "textmsg(num_barreno,pos_barreno)"
            textmsg(num_barreno,pos_barreno)
          end
          $ 1400 "Poses_taladrado≔pose_add(get_actual_tcp_pose(), bajada_broca)"
          global Poses_taladrado= pose_add ( get_actual_tcp_pose (), bajada_broca)
          $ 1401 "Poses_taladrado" "breakAfter"
          movel(Poses_taladrado, a=0.01, v=0.01)
          $ 1402 "bajada_broca≔pose_add(bajada_broca, p[0,0,0.009,0,0,0])"
          global bajada_broca= pose_add (bajada_broca, p[0,0,0.009,0,0,0])
          Loop_74 = Loop_74 + 1
        end
